// TIA Portal V15.1 export
// export: Created 2024-06-21T08:41:01.4306107Z, ExportSetting WithDefaults, DisplayName Totally Integrated Automation Portal, DisplayVersion V15.1 Update 5, DisplayName TIA Portal Openness, DisplayVersion V15.1 Update 5, DisplayName SINAMICS Startdrive Advanced, DisplayVersion V15.1, DisplayName G130, G150, S120, S150, SINAMICS MV, S210, DisplayVersion V15.1, DisplayName G110M, G120, G120C, G120D, G120P, DisplayVersion V15.1, DisplayName STEP 7 Professional, DisplayVersion V15.1 Update 5, DisplayName STEP 7 Safety, DisplayVersion V15.1, DisplayName WinCC Professional, DisplayVersion V15.1 Update 5, DisplayName SIMATIC Visualization Architect, DisplayVersion V15.1
FUNCTION_BLOCK "LModeSelector"   // FB1002, FBD
TITLE = LModeSelector
{ S7_Optimized_Access := 'FALSE' }
AUTHOR : VCC
FAMILY : Control
NAME : ModeSel
VERSION : 1.0
// ================================================================================
// This module handles that only one mode is selected in the modezon, it also 
// handle interlocking between the HMIs. Each modezone can have 5 HMI.
// ================================================================================
// stored: AutoNumber false, IsIECCheckEnabled false, SetENOAutomatically False, UDAEnableTagReadback false
   VAR_INPUT
      I_NumHMI { ExternalAccessible := 'False'; ExternalVisible := 'False'; ExternalWritable := 'False'} : Int;   // Number of HMI used in the modezon
      I_LockManualTime { ExternalAccessible := 'False'; ExternalVisible := 'False'; ExternalWritable := 'False'} : Int;   // The number of seconds that Lock Manual shall be active
      I_StartPB { ExternalAccessible := 'False'; ExternalVisible := 'False'; ExternalWritable := 'False'} : Bool;   // Summary of Start buttons
      I_AlarmResetPB { ExternalAccessible := 'False'; ExternalVisible := 'False'; ExternalWritable := 'False'} : Bool;   // Summary of Alarm reset buttons
      I_SafetyNotOk { ExternalAccessible := 'False'; ExternalVisible := 'False'; ExternalWritable := 'False'} : Bool;   // Safety is not ok
      I_FailSafeResetAck { ExternalAccessible := 'False'; ExternalVisible := 'False'; ExternalWritable := 'False'} : Bool;   // F_Ack_Op FB in safety program is requesting value 9 on FailSafeReset output
      I_FailSafeAckID { ExternalAccessible := 'False'; ExternalVisible := 'False'; ExternalWritable := 'False'} : Int;   // F_Ack ID
      I_AllHMIAutoSel { ExternalAccessible := 'False'; ExternalVisible := 'False'; ExternalWritable := 'False'} : Bool;   // All HMI to Auto Selected
      I_HMI1ForceMan { ExternalAccessible := 'False'; ExternalVisible := 'False'; ExternalWritable := 'False'} : Bool;   // Forced manual selected on HMI1
      I_HMI1SetPB { ExternalAccessible := 'False'; ExternalVisible := 'False'; ExternalWritable := 'False'} : Bool;   // Set PB activated on HMI1
      I_HMI1ResetPB { ExternalAccessible := 'False'; ExternalVisible := 'False'; ExternalWritable := 'False'} : Bool;   // Reset PB activated on HMI1
      I_HMI1StartPB { ExternalAccessible := 'False'; ExternalVisible := 'False'; ExternalWritable := 'False'} : Bool;   // Start PB activated on HMI1
      I_HMI1AlarmResetPB { ExternalAccessible := 'False'; ExternalVisible := 'False'; ExternalWritable := 'False'} : Bool;   // AlarmReset PB activated on HMI1
      I_HMI2ForceMan { ExternalAccessible := 'False'; ExternalVisible := 'False'; ExternalWritable := 'False'} : Bool;   // Forced manual selected on HMI2
      I_HMI2SetPB { ExternalAccessible := 'False'; ExternalVisible := 'False'; ExternalWritable := 'False'} : Bool;   // Set PB activated on HMI2
      I_HMI2ResetPB { ExternalAccessible := 'False'; ExternalVisible := 'False'; ExternalWritable := 'False'} : Bool;   // Reset PB activated on HMI2
      I_HMI2StartPB { ExternalAccessible := 'False'; ExternalVisible := 'False'; ExternalWritable := 'False'} : Bool;   // Start PB activated on HMI2
      I_HMI2AlarmResetPB { ExternalAccessible := 'False'; ExternalVisible := 'False'; ExternalWritable := 'False'} : Bool;   // AlarmReset PB activated on HMI2
      I_HMI3ForceMan { ExternalAccessible := 'False'; ExternalVisible := 'False'; ExternalWritable := 'False'} : Bool;   // Forced manual selected on HMI3
      I_HMI3SetPB { ExternalAccessible := 'False'; ExternalVisible := 'False'; ExternalWritable := 'False'} : Bool;   // Set PB activated on HMI3
      I_HMI3ResetPB { ExternalAccessible := 'False'; ExternalVisible := 'False'; ExternalWritable := 'False'} : Bool;   // Reset PB activated on HMI3
      I_HMI3StartPB { ExternalAccessible := 'False'; ExternalVisible := 'False'; ExternalWritable := 'False'} : Bool;   // Start PB activated on HMI
      I_HMI3AlarmResetPB { ExternalAccessible := 'False'; ExternalVisible := 'False'; ExternalWritable := 'False'} : Bool;   // AlarmReset PB activated on HMI3
      I_HMI4ForceMan { ExternalAccessible := 'False'; ExternalVisible := 'False'; ExternalWritable := 'False'} : Bool;   // Forced manual selected on HMI4
      I_HMI4SetPB { ExternalAccessible := 'False'; ExternalVisible := 'False'; ExternalWritable := 'False'} : Bool;   // Set PB activated on HMI4
      I_HMI4ResetPB { ExternalAccessible := 'False'; ExternalVisible := 'False'; ExternalWritable := 'False'} : Bool;   // Reset PB activated on HMI4
      I_HMI4StartPB { ExternalAccessible := 'False'; ExternalVisible := 'False'; ExternalWritable := 'False'} : Bool;   // Start PB activated on HMI4
      I_HMI4AlarmResetPB { ExternalAccessible := 'False'; ExternalVisible := 'False'; ExternalWritable := 'False'} : Bool;   // AlarmReset PB activated on HMI4
      I_HMI5ForceMan { ExternalAccessible := 'False'; ExternalVisible := 'False'; ExternalWritable := 'False'} : Bool;   // Forced manual selected on HMI5
      I_HMI5SetPB { ExternalAccessible := 'False'; ExternalVisible := 'False'; ExternalWritable := 'False'} : Bool;   // Set PB activated on HMI5
      I_HMI5ResetPB { ExternalAccessible := 'False'; ExternalVisible := 'False'; ExternalWritable := 'False'} : Bool;   // Reset PB activated on HMI5
      I_HMI5StartPB { ExternalAccessible := 'False'; ExternalVisible := 'False'; ExternalWritable := 'False'} : Bool;   // Start PB activated on HMI5
      I_HMI5AlarmResetPB { ExternalAccessible := 'False'; ExternalVisible := 'False'; ExternalWritable := 'False'} : Bool;   // AlarmReset PB activated on HMI5
   END_VAR
   VAR_OUTPUT
      O_AutoSel { ExternalAccessible := 'False'; ExternalVisible := 'False'; ExternalWritable := 'False'} : Bool;   // Auto selected
      O_AllAutoSel { ExternalAccessible := 'False'; ExternalVisible := 'False'; ExternalWritable := 'False'} : Bool;   // All objects in Auto selected
      O_StepSel { ExternalAccessible := 'False'; ExternalVisible := 'False'; ExternalWritable := 'False'} : Bool;   // Step selected
      O_HomeRunSel { ExternalAccessible := 'False'; ExternalVisible := 'False'; ExternalWritable := 'False'} : Bool;   // Homerun selected
      O_ManualSel { ExternalAccessible := 'False'; ExternalVisible := 'False'; ExternalWritable := 'False'} : Bool;   // Manual selected
      O_ForcedManActSel { ExternalAccessible := 'False'; ExternalVisible := 'False'; ExternalWritable := 'False'} : Bool;   // Forced manual selected
      O_PBSetSel { ExternalAccessible := 'False'; ExternalVisible := 'False'; ExternalWritable := 'False'} : Bool;   // Set selected
      O_PBResetSel { ExternalAccessible := 'False'; ExternalVisible := 'False'; ExternalWritable := 'False'} : Bool;   // Reset selected
      O_StartPBSel { ExternalAccessible := 'False'; ExternalVisible := 'False'; ExternalWritable := 'False'} : Bool;   // Start is activated
      O_AlarmResetPBSel { ExternalAccessible := 'False'; ExternalVisible := 'False'; ExternalWritable := 'False'} : Bool;   // Alarm reset is activated
      O_ResetTMSel { ExternalAccessible := 'False'; ExternalVisible := 'False'; ExternalWritable := 'False'} : Bool;   // Reset transport memory
      O_ResetSeqSel { ExternalAccessible := 'False'; ExternalVisible := 'False'; ExternalWritable := 'False'} : Bool;   // Reset squence
      O_CycleFinishedSel { ExternalAccessible := 'False'; ExternalVisible := 'False'; ExternalWritable := 'False'} : Bool;   // Cycle finished selected
      O_HomeRunRedoSel { ExternalAccessible := 'False'; ExternalVisible := 'False'; ExternalWritable := 'False'} : Bool;   // Redo after Homerun selected
      O_HomeRunWorkDoneSel { ExternalAccessible := 'False'; ExternalVisible := 'False'; ExternalWritable := 'False'} : Bool;   // WorkDone after Homerun selected
   END_VAR
   VAR_IN_OUT
      IO_FailsafeReset { ExternalAccessible := 'False'; ExternalVisible := 'False'; ExternalWritable := 'False'} : Int;   // Number to Failsafe to reset safety
   END_VAR
   VAR DB_SPECIFIC
      H_HMIHomeRunModeCmd : Word;   // Homerun Mode commands from HMI
      H_Anim : Word;   // Animation for HMI
      H_ActiveHMI : Int;   // Active HMI
      H_NameActiveHMI : String[25];   // Name of the Active HMI
      H_LockManTime : Int;   // Lock manual time
      H_HMI1ModeCmd : Word;   // Mode commands from HMI1
      H_HMI2ModeCmd : Word;   // Mode commands from HMI2
      H_HMI3ModeCmd : Word;   // Mode commands from HMI3
      H_HMI4ModeCmd : Word;   // Mode commands from HMI4
      H_HMI5ModeCmd : Word;   // Mode commands from HMI5. For operator panels, no S7_m_c
      HMI1AutoSel { ExternalAccessible := 'False'; ExternalVisible := 'False'; ExternalWritable := 'False'} : Bool;   // Auto selected on HMI1
      HMI1StepSel { ExternalAccessible := 'False'; ExternalVisible := 'False'; ExternalWritable := 'False'} : Bool;   // Step selected on HMI1
      HMI1HomeRunSel { ExternalAccessible := 'False'; ExternalVisible := 'False'; ExternalWritable := 'False'} : Bool;   // Homerun selected on HMI1
      HMI1ManualSel { ExternalAccessible := 'False'; ExternalVisible := 'False'; ExternalWritable := 'False'} : Bool;   // Manual selected on HMI1
      HMI1LockManual { ExternalAccessible := 'False'; ExternalVisible := 'False'; ExternalWritable := 'False'} : Bool;   // Lock manual for HMI1
      HMI1AllHMIAutoSel { ExternalAccessible := 'False'; ExternalVisible := 'False'; ExternalWritable := 'False'} : Bool;   // All HMI Auto selected on HMI1
      HMI1Start { ExternalAccessible := 'False'; ExternalVisible := 'False'; ExternalWritable := 'False'} : Bool;   // Start on HMI1
      HMI1AlarmReset { ExternalAccessible := 'False'; ExternalVisible := 'False'; ExternalWritable := 'False'} : Bool;   // AlarmReset on HMI1
      HMI1ResetTM { ExternalAccessible := 'False'; ExternalVisible := 'False'; ExternalWritable := 'False'} : Bool;   // Reset transport memory from HMI1
      HMI1ResetSeq { ExternalAccessible := 'False'; ExternalVisible := 'False'; ExternalWritable := 'False'} : Bool;   // Reset sequence from HMI1
      HMI1CycleFinished { ExternalAccessible := 'False'; ExternalVisible := 'False'; ExternalWritable := 'False'} : Bool;   // Cycle Finished from HMI1
      HMI1AlarmResetAck { ExternalAccessible := 'False'; ExternalVisible := 'False'; ExternalWritable := 'False'} : Bool;   // Alarm Reset acknowledge from HMI1
      HMI2AutoSel { ExternalAccessible := 'False'; ExternalVisible := 'False'; ExternalWritable := 'False'} : Bool;   // Auto selected on HMI2
      HMI2StepSel { ExternalAccessible := 'False'; ExternalVisible := 'False'; ExternalWritable := 'False'} : Bool;   // Step selected on HMI2
      HMI2HomeRunSel { ExternalAccessible := 'False'; ExternalVisible := 'False'; ExternalWritable := 'False'} : Bool;   // Homerun selected on HMI2
      HMI2ManualSel { ExternalAccessible := 'False'; ExternalVisible := 'False'; ExternalWritable := 'False'} : Bool;   // Manual selected on HMI2
      HMI2LockManual { ExternalAccessible := 'False'; ExternalVisible := 'False'; ExternalWritable := 'False'} : Bool;   // Lock manual for HMI2
      HMI2AllHMIAutoSel { ExternalAccessible := 'False'; ExternalVisible := 'False'; ExternalWritable := 'False'} : Bool;   // All HMI Auto selected on HMI2
      HMI2Start { ExternalAccessible := 'False'; ExternalVisible := 'False'; ExternalWritable := 'False'} : Bool;   // Start on HMI2
      HMI2AlarmReset { ExternalAccessible := 'False'; ExternalVisible := 'False'; ExternalWritable := 'False'} : Bool;   // AlarmReset on HMI2
      HMI2ResetTM { ExternalAccessible := 'False'; ExternalVisible := 'False'; ExternalWritable := 'False'} : Bool;   // Reset transport memory from HMI2
      HMI2ResetSeq { ExternalAccessible := 'False'; ExternalVisible := 'False'; ExternalWritable := 'False'} : Bool;   // Reset sequence from HMI2
      HMI2CycleFinished { ExternalAccessible := 'False'; ExternalVisible := 'False'; ExternalWritable := 'False'} : Bool;   // Cycle Finished from HMI2
      HMI2AlarmResetAck { ExternalAccessible := 'False'; ExternalVisible := 'False'; ExternalWritable := 'False'} : Bool;   // Alarm Reset acknowledge from HMI2
      HMI3AutoSel { ExternalAccessible := 'False'; ExternalVisible := 'False'; ExternalWritable := 'False'} : Bool;   // Auto selected on HMI3
      HMI3StepSel { ExternalAccessible := 'False'; ExternalVisible := 'False'; ExternalWritable := 'False'} : Bool;   // Step selected on HMI3
      HMI3HomeRunSel { ExternalAccessible := 'False'; ExternalVisible := 'False'; ExternalWritable := 'False'} : Bool;   // Homerun selected on HMI3
      HMI3ManualSel { ExternalAccessible := 'False'; ExternalVisible := 'False'; ExternalWritable := 'False'} : Bool;   // Manual selected on HMI3
      HMI3LockManual { ExternalAccessible := 'False'; ExternalVisible := 'False'; ExternalWritable := 'False'} : Bool;   // Lock manual for HMI3
      HMI3AllHMIAutoSel { ExternalAccessible := 'False'; ExternalVisible := 'False'; ExternalWritable := 'False'} : Bool;   // All HMI Auto selected on HMI3
      HMI3Start { ExternalAccessible := 'False'; ExternalVisible := 'False'; ExternalWritable := 'False'} : Bool;   // Start on HMI3
      HMI3AlarmReset { ExternalAccessible := 'False'; ExternalVisible := 'False'; ExternalWritable := 'False'} : Bool;   // AlarmReset on HMI3
      HMI3ResetTM { ExternalAccessible := 'False'; ExternalVisible := 'False'; ExternalWritable := 'False'} : Bool;   // Reset transport memory from HMI3
      HMI3ResetSeq { ExternalAccessible := 'False'; ExternalVisible := 'False'; ExternalWritable := 'False'} : Bool;   // Reset sequence from HMI3
      HMI3CycleFinished { ExternalAccessible := 'False'; ExternalVisible := 'False'; ExternalWritable := 'False'} : Bool;   // Cycle Finished from HMI3
      HMI3AlarmResetAck { ExternalAccessible := 'False'; ExternalVisible := 'False'; ExternalWritable := 'False'} : Bool;   // Alarm Reset acknowledge from 3
      HMI4AutoSel { ExternalAccessible := 'False'; ExternalVisible := 'False'; ExternalWritable := 'False'} : Bool;   // Auto selected on HMI4
      HMI4StepSel { ExternalAccessible := 'False'; ExternalVisible := 'False'; ExternalWritable := 'False'} : Bool;   // Step selected on HMI4
      HMI4HomeRunSel { ExternalAccessible := 'False'; ExternalVisible := 'False'; ExternalWritable := 'False'} : Bool;   // Homerun selected on HMI4
      HMI4ManualSel { ExternalAccessible := 'False'; ExternalVisible := 'False'; ExternalWritable := 'False'} : Bool;   // Manual selected on HMI4
      HMI4LockManual { ExternalAccessible := 'False'; ExternalVisible := 'False'; ExternalWritable := 'False'} : Bool;   // Lock manual for HMI4
      HMI4AllHMIAutoSel { ExternalAccessible := 'False'; ExternalVisible := 'False'; ExternalWritable := 'False'} : Bool;   // All HMI Auto selected on HMI4
      HMI4Start { ExternalAccessible := 'False'; ExternalVisible := 'False'; ExternalWritable := 'False'} : Bool;   // Start on HMI4
      HMI4AlarmReset { ExternalAccessible := 'False'; ExternalVisible := 'False'; ExternalWritable := 'False'} : Bool;   // AlarmReset on HMI4
      HMI4ResetTM { ExternalAccessible := 'False'; ExternalVisible := 'False'; ExternalWritable := 'False'} : Bool;   // Reset transport memory from HMI4
      HMI4ResetSeq { ExternalAccessible := 'False'; ExternalVisible := 'False'; ExternalWritable := 'False'} : Bool;   // Reset sequence from HMI4
      HMI4CycleFinished { ExternalAccessible := 'False'; ExternalVisible := 'False'; ExternalWritable := 'False'} : Bool;   // Cycle Finished from HMI4
      HMI4AlarmResetAck { ExternalAccessible := 'False'; ExternalVisible := 'False'; ExternalWritable := 'False'} : Bool;   // Alarm Reset acknowledge from HMI4
      HMI5AutoSel { ExternalAccessible := 'False'; ExternalVisible := 'False'; ExternalWritable := 'False'} : Bool;   // Auto selected on HMI5
      HMI5StepSel { ExternalAccessible := 'False'; ExternalVisible := 'False'; ExternalWritable := 'False'} : Bool;   // Step selected on HMI5
      HMI5HomeRunSel { ExternalAccessible := 'False'; ExternalVisible := 'False'; ExternalWritable := 'False'} : Bool;   // Homerun selected on HMI5
      HMI5ManualSel { ExternalAccessible := 'False'; ExternalVisible := 'False'; ExternalWritable := 'False'} : Bool;   // Manual selected on HMI5
      HMI5LockManual { ExternalAccessible := 'False'; ExternalVisible := 'False'; ExternalWritable := 'False'} : Bool;   // Lock manual for HMI5
      HMI5AllHMIAutoSel { ExternalAccessible := 'False'; ExternalVisible := 'False'; ExternalWritable := 'False'} : Bool;   // All HMI Auto selected on HMI5
      HMI5Start { ExternalAccessible := 'False'; ExternalVisible := 'False'; ExternalWritable := 'False'} : Bool;   // Start on HMI5
      HMI5AlarmReset { ExternalAccessible := 'False'; ExternalVisible := 'False'; ExternalWritable := 'False'} : Bool;   // AlarmReset on HMI5
      HMI5ResetTM { ExternalAccessible := 'False'; ExternalVisible := 'False'; ExternalWritable := 'False'} : Bool;   // Reset transport memory from HMI5
      HMI5ResetSeq { ExternalAccessible := 'False'; ExternalVisible := 'False'; ExternalWritable := 'False'} : Bool;   // Reset sequence from HMI5
      HMI5CycleFinished { ExternalAccessible := 'False'; ExternalVisible := 'False'; ExternalWritable := 'False'} : Bool;   // Cycle Finished from HMI5
      HMI5AlarmResetAck { ExternalAccessible := 'False'; ExternalVisible := 'False'; ExternalWritable := 'False'} : Bool;   // Alarm Reset acknowledge from HMI5
      HMIHomeRunRedo { ExternalAccessible := 'False'; ExternalVisible := 'False'; ExternalWritable := 'False'} : Bool;   // Redo after homerun from HMI
      HMIHomeRunWorkDone { ExternalAccessible := 'False'; ExternalVisible := 'False'; ExternalWritable := 'False'} : Bool;   // WorkDone after homerun from HMI
      LockManualTimeout { ExternalAccessible := 'False'; ExternalVisible := 'False'; ExternalWritable := 'False'} : Bool;   // Lock manual button timeout
      AllHmiAutoSel { ExternalAccessible := 'False'; ExternalVisible := 'False'; ExternalWritable := 'False'} : Bool;   // All Hmi Auto selected
      AlarmResetPBSel { ExternalAccessible := 'False'; ExternalVisible := 'False'; ExternalWritable := 'False'} : Bool;   // Alarm reset is activated
      AlarmResetPBSelReset { ExternalAccessible := 'False'; ExternalVisible := 'False'; ExternalWritable := 'False'} : Bool;   // Reset AlarmResetPBSel after predefined time
      AlarmResetPBSelResetPE { ExternalAccessible := 'False'; ExternalVisible := 'False'; ExternalWritable := 'False'} : Bool;   // Positive edge of AlarmResetPbSelReset
      FailSafeReset6Pulse { ExternalAccessible := 'False'; ExternalVisible := 'False'; ExternalWritable := 'False'} : Bool;   // Pulse to set value 6 on FailSafeReset Output
      FailSafeReset9Pulse { ExternalAccessible := 'False'; ExternalVisible := 'False'; ExternalWritable := 'False'} : Bool;   // Pulse to set value 9 on FailSafeReset Output
      ResetAlarmAckMemPulse { ExternalAccessible := 'False'; ExternalVisible := 'False'; ExternalWritable := 'False'} : Bool;   // Pulse to reset AlarmResetAckMem on negative edge of I_FailSafeResetAck
      AlarmResetAckMem { ExternalAccessible := 'False'; ExternalVisible := 'False'; ExternalWritable := 'False'} : Bool;   // memory : Pushbutton AlarmResetAck has been pushed on HMI
      StartPBSel { ExternalAccessible := 'False'; ExternalVisible := 'False'; ExternalWritable := 'False'} : Bool;   // Summary of the Start push buttons
      AutoSel { ExternalAccessible := 'False'; ExternalVisible := 'False'; ExternalWritable := 'False'} : Bool;   // Auto selected
      HMIStartPE { ExternalAccessible := 'False'; ExternalVisible := 'False'; ExternalWritable := 'False'} : Bool;   // Positive edge on start button from HMI
      HMIResetTMPE { ExternalAccessible := 'False'; ExternalVisible := 'False'; ExternalWritable := 'False'} : Bool;   // Positive edge on ResetTM button from HMI
      HMIResetSeqPE { ExternalAccessible := 'False'; ExternalVisible := 'False'; ExternalWritable := 'False'} : Bool;   // Positive edge on ResetSeq button from HMI
      HMIAlarmResetAckPE { ExternalAccessible := 'False'; ExternalVisible := 'False'; ExternalWritable := 'False'} : Bool;   // Positive edge on AlarmResetAck button from HMI
      HMILockManualPE { ExternalAccessible := 'False'; ExternalVisible := 'False'; ExternalWritable := 'False'} : Bool;   // Positive edge on LockManual button from HMI
      PBSetSel { ExternalAccessible := 'False'; ExternalVisible := 'False'; ExternalWritable := 'False'} : Bool;   // Set selected
      PBResetSel { ExternalAccessible := 'False'; ExternalVisible := 'False'; ExternalWritable := 'False'} : Bool;   // Reset selected
      CheckHMIActive { ExternalAccessible := 'False'; ExternalVisible := 'False'; ExternalWritable := 'False'} : Bool;   // Check Active HMI
      FailsafeReset { ExternalAccessible := 'False'; ExternalVisible := 'False'; ExternalWritable := 'False'} : Int;   // Number to Failsafe to reset safety
      ActiveHMI { ExternalAccessible := 'False'; ExternalVisible := 'False'; ExternalWritable := 'False'} : Int;   // Help memory for Active HMI
      LockManualSec { ExternalAccessible := 'False'; ExternalVisible := 'False'; ExternalWritable := 'False'} : DInt;   // Lock manual on for xxx milliesec
      LockManualMillieSec { ExternalAccessible := 'False'; ExternalVisible := 'False'; ExternalWritable := 'False'} : DInt;   // Converted value
      TimerLockManValue { ExternalAccessible := 'False'; ExternalVisible := 'False'; ExternalWritable := 'False'} : DInt;   // Timer value
   END_VAR
   VAR
      TimerLockMan { ExternalAccessible := 'False'; ExternalVisible := 'False'; ExternalWritable := 'False'; S7_SetPoint := 'True'} : "LTimer";   // Timer on Lock manual
      TimerAlarmResetPB { ExternalAccessible := 'False'; ExternalVisible := 'False'; ExternalWritable := 'False'; S7_SetPoint := 'True'} : "LTimer";   // Timer on alarm reset
   END_VAR
   VAR DB_SPECIFIC
      CheckActiveHMI { ExternalAccessible := 'False'; ExternalVisible := 'False'; ExternalWritable := 'False'; S7_SetPoint := 'True'} : TP_TIME;   // Timer
      CheckActiveHMI_1 { ExternalAccessible := 'False'; ExternalVisible := 'False'; ExternalWritable := 'False'; S7_SetPoint := 'True'} : TP_TIME;   // Timer
      CheckActiveHMI_2 { ExternalAccessible := 'False'; ExternalVisible := 'False'; ExternalWritable := 'False'; S7_SetPoint := 'True'} : TON_TIME;   // Timer
      CheckActiveHMI_3 { ExternalAccessible := 'False'; ExternalVisible := 'False'; ExternalWritable := 'False'; S7_SetPoint := 'True'} : TON_TIME;   // Timer
   END_VAR
   VAR_TEMP
      PHMI1AutoSel : Bool;   // Pulse Auto selected HMI1
      PHMI2AutoSel : Bool;   // Pulse Auto selected HMI2
      PHMI3AutoSel : Bool;   // Pulse Auto selected HMI3
      PHMI4AutoSel : Bool;   // Pulse Auto selected HMI4
      PHMI5AutoSel : Bool;   // Pulse Auto selected HMI5
      LockManualTime : Int;   // Lock manual time
      LockManualTimeInt : Int;   // Lock manual time
      LockManualTimeDInt : DInt;   // Lock manual time
   END_VAR
   VAR_TEMP   // added for the SCL form of the ladder/FBD networks
      _w1 : Bool;
      _w2 : Bool;
      _w3 : Bool;
      _w4 : Bool;
      _w5 : Bool;
   END_VAR
BEGIN

REGION Network 1: **** 1 - Inputs **** Extract the modeselection from HMI 1
   // Extract the modeselection from HMI 1
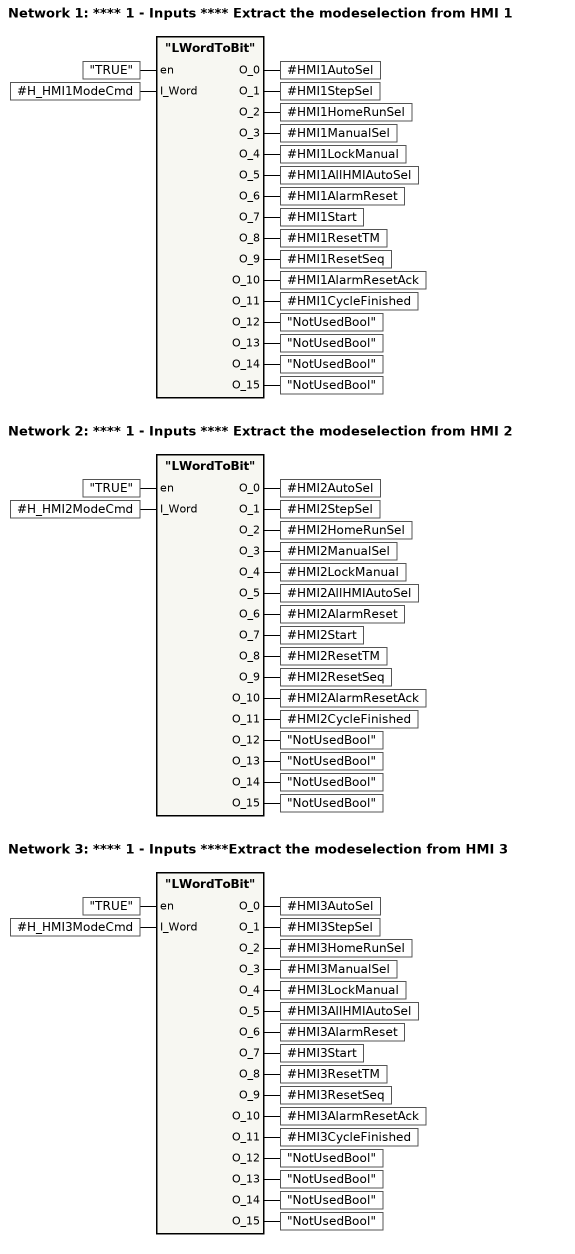
   IF "TRUE" THEN
       "LWordToBit"(I_Word := #H_HMI1ModeCmd,
                    O_0 => #HMI1AutoSel,
                    O_1 => #HMI1StepSel,
                    O_2 => #HMI1HomeRunSel,
                    O_3 => #HMI1ManualSel,
                    O_4 => #HMI1LockManual,
                    O_5 => #HMI1AllHMIAutoSel,
                    O_6 => #HMI1AlarmReset,
                    O_7 => #HMI1Start,
                    O_8 => #HMI1ResetTM,
                    O_9 => #HMI1ResetSeq,
                    O_10 => #HMI1AlarmResetAck,
                    O_11 => #HMI1CycleFinished,
                    O_12 => "NotUsedBool",
                    O_13 => "NotUsedBool",
                    O_14 => "NotUsedBool",
                    O_15 => "NotUsedBool");
   END_IF;
END_REGION

REGION Network 2: **** 1 - Inputs **** Extract the modeselection from HMI 2
   // Extract the modeselection from HMI 2
   IF "TRUE" THEN
       "LWordToBit"(I_Word := #H_HMI2ModeCmd,
                    O_0 => #HMI2AutoSel,
                    O_1 => #HMI2StepSel,
                    O_2 => #HMI2HomeRunSel,
                    O_3 => #HMI2ManualSel,
                    O_4 => #HMI2LockManual,
                    O_5 => #HMI2AllHMIAutoSel,
                    O_6 => #HMI2AlarmReset,
                    O_7 => #HMI2Start,
                    O_8 => #HMI2ResetTM,
                    O_9 => #HMI2ResetSeq,
                    O_10 => #HMI2AlarmResetAck,
                    O_11 => #HMI2CycleFinished,
                    O_12 => "NotUsedBool",
                    O_13 => "NotUsedBool",
                    O_14 => "NotUsedBool",
                    O_15 => "NotUsedBool");
   END_IF;
END_REGION

REGION Network 3: **** 1 - Inputs ****Extract the modeselection from HMI 3
   // Extract the modeselection from HMI 3
   IF "TRUE" THEN
       "LWordToBit"(I_Word := #H_HMI3ModeCmd,
                    O_0 => #HMI3AutoSel,
                    O_1 => #HMI3StepSel,
                    O_2 => #HMI3HomeRunSel,
                    O_3 => #HMI3ManualSel,
                    O_4 => #HMI3LockManual,
                    O_5 => #HMI3AllHMIAutoSel,
                    O_6 => #HMI3AlarmReset,
                    O_7 => #HMI3Start,
                    O_8 => #HMI3ResetTM,
                    O_9 => #HMI3ResetSeq,
                    O_10 => #HMI3AlarmResetAck,
                    O_11 => #HMI3CycleFinished,
                    O_12 => "NotUsedBool",
                    O_13 => "NotUsedBool",
                    O_14 => "NotUsedBool",
                    O_15 => "NotUsedBool");
   END_IF;
END_REGION

REGION Network 4: **** 1 - Inputs **** Extract the modeselection from HMI 4
   // Extract the modeselection from HMI 4
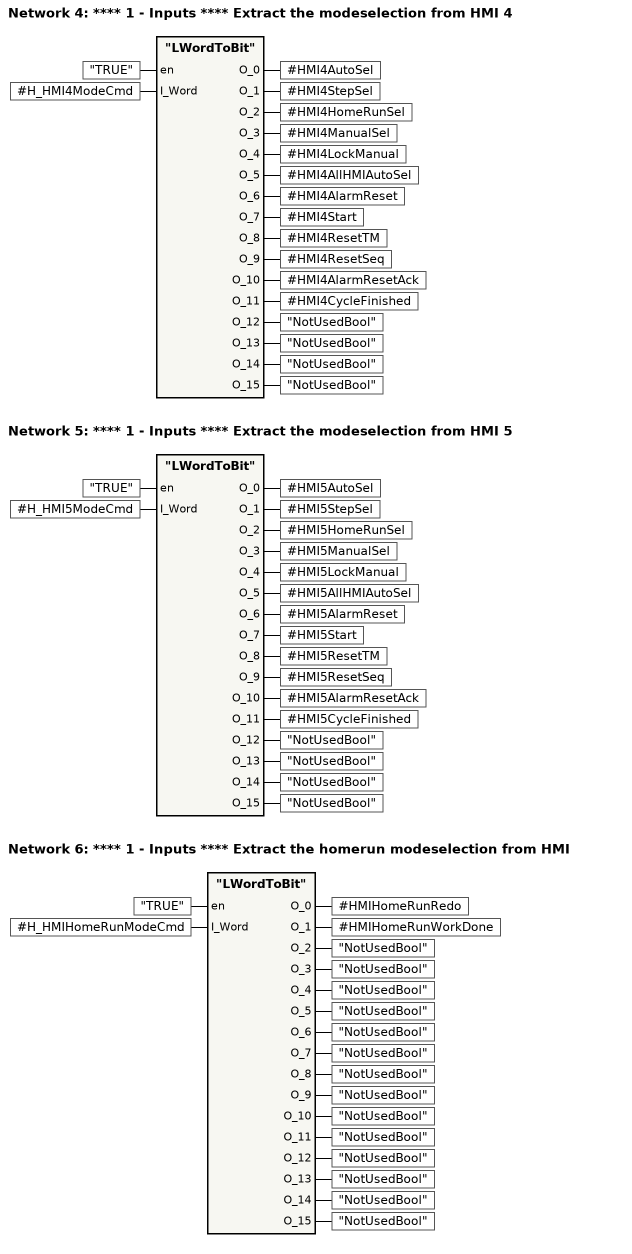
   IF "TRUE" THEN
       "LWordToBit"(I_Word := #H_HMI4ModeCmd,
                    O_0 => #HMI4AutoSel,
                    O_1 => #HMI4StepSel,
                    O_2 => #HMI4HomeRunSel,
                    O_3 => #HMI4ManualSel,
                    O_4 => #HMI4LockManual,
                    O_5 => #HMI4AllHMIAutoSel,
                    O_6 => #HMI4AlarmReset,
                    O_7 => #HMI4Start,
                    O_8 => #HMI4ResetTM,
                    O_9 => #HMI4ResetSeq,
                    O_10 => #HMI4AlarmResetAck,
                    O_11 => #HMI4CycleFinished,
                    O_12 => "NotUsedBool",
                    O_13 => "NotUsedBool",
                    O_14 => "NotUsedBool",
                    O_15 => "NotUsedBool");
   END_IF;
END_REGION

REGION Network 5: **** 1 - Inputs **** Extract the modeselection from HMI 5
   // Extract the modeselection from HMI 5
   IF "TRUE" THEN
       "LWordToBit"(I_Word := #H_HMI5ModeCmd,
                    O_0 => #HMI5AutoSel,
                    O_1 => #HMI5StepSel,
                    O_2 => #HMI5HomeRunSel,
                    O_3 => #HMI5ManualSel,
                    O_4 => #HMI5LockManual,
                    O_5 => #HMI5AllHMIAutoSel,
                    O_6 => #HMI5AlarmReset,
                    O_7 => #HMI5Start,
                    O_8 => #HMI5ResetTM,
                    O_9 => #HMI5ResetSeq,
                    O_10 => #HMI5AlarmResetAck,
                    O_11 => #HMI5CycleFinished,
                    O_12 => "NotUsedBool",
                    O_13 => "NotUsedBool",
                    O_14 => "NotUsedBool",
                    O_15 => "NotUsedBool");
   END_IF;
END_REGION

REGION Network 6: **** 1 - Inputs **** Extract the homerun modeselection from HMI
   // Extract the homerun modeselection from HMI
   IF "TRUE" THEN
       "LWordToBit"(I_Word := #H_HMIHomeRunModeCmd,
                    O_0 => #HMIHomeRunRedo,
                    O_1 => #HMIHomeRunWorkDone,
                    O_2 => "NotUsedBool",
                    O_3 => "NotUsedBool",
                    O_4 => "NotUsedBool",
                    O_5 => "NotUsedBool",
                    O_6 => "NotUsedBool",
                    O_7 => "NotUsedBool",
                    O_8 => "NotUsedBool",
                    O_9 => "NotUsedBool",
                    O_10 => "NotUsedBool",
                    O_11 => "NotUsedBool",
                    O_12 => "NotUsedBool",
                    O_13 => "NotUsedBool",
                    O_14 => "NotUsedBool",
                    O_15 => "NotUsedBool");
   END_IF;
END_REGION

REGION Network 7: **** 1 - Inputs **** All HMI Auto selected
   // All HMI Auto selected
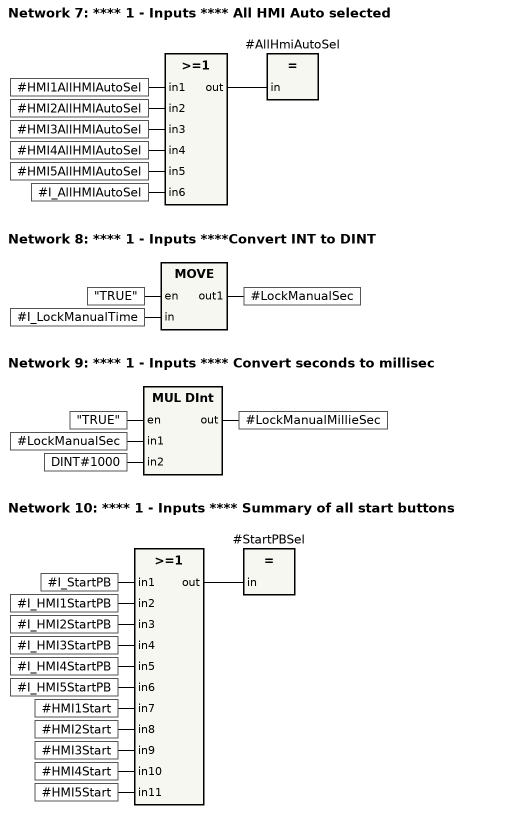
   #AllHmiAutoSel := #HMI1AllHMIAutoSel OR #HMI2AllHMIAutoSel OR #HMI3AllHMIAutoSel OR #HMI4AllHMIAutoSel OR #HMI5AllHMIAutoSel OR #I_AllHMIAutoSel;
END_REGION

REGION Network 8: **** 1 - Inputs ****Convert INT to DINT
   // Convert INT to DINT
   IF "TRUE" THEN #LockManualSec := #I_LockManualTime; END_IF;
END_REGION

REGION Network 9: **** 1 - Inputs **** Convert seconds to millisec
   // Convert seconds to millisec
   IF "TRUE" THEN #LockManualMillieSec := #LockManualSec * DINT#1000; END_IF;
END_REGION

REGION Network 10: **** 1 - Inputs **** Summary of all start buttons
   // Summary of all start buttons
   #StartPBSel := #I_StartPB OR #I_HMI1StartPB OR #I_HMI2StartPB OR #I_HMI3StartPB OR #I_HMI4StartPB OR #I_HMI5StartPB OR #HMI1Start OR #HMI2Start OR #HMI3Start OR #HMI4Start OR #HMI5Start;
END_REGION

REGION Network 11: **** 1 - Inputs **** Reset Start button from HMI
   // Reset Start button from HMI
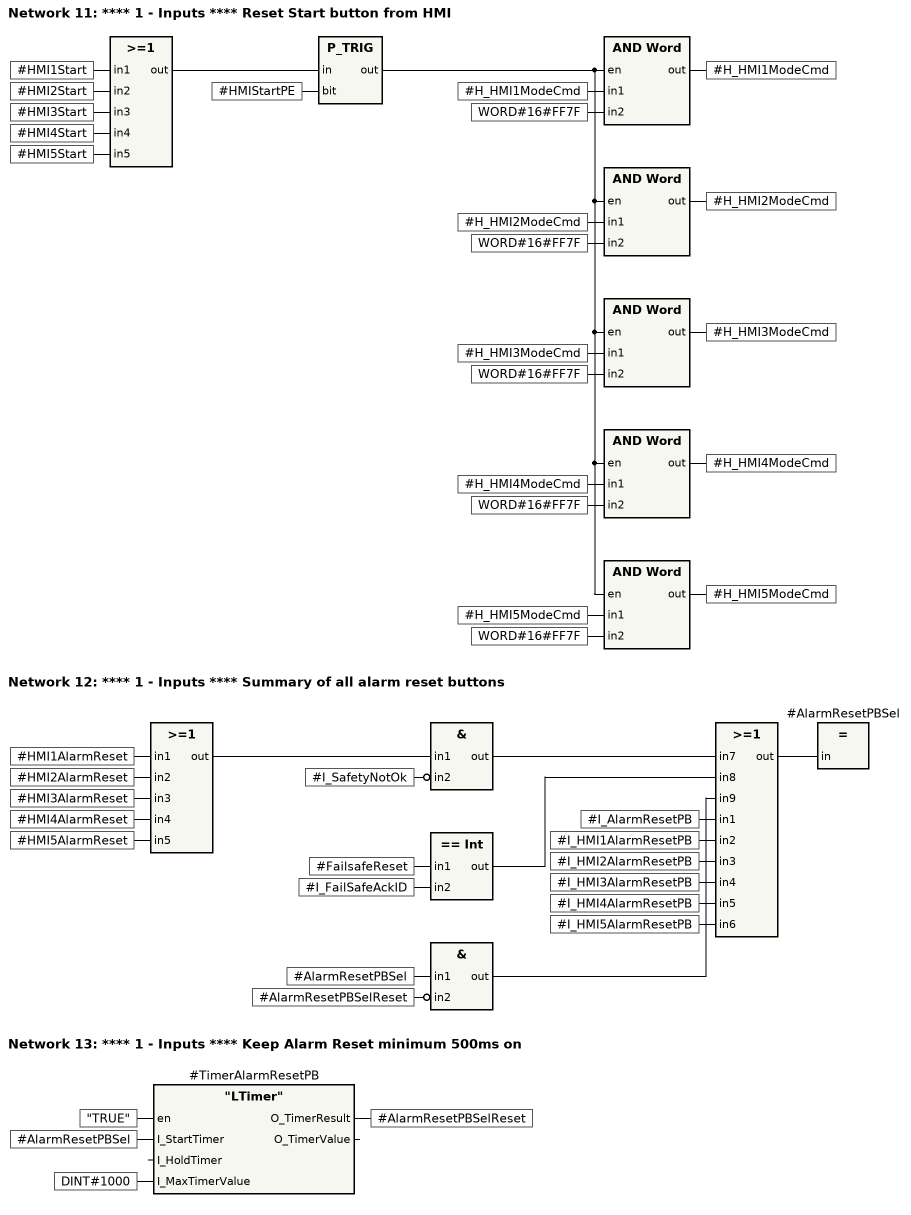
   #_w1 := #HMI1Start OR #HMI2Start OR #HMI3Start OR #HMI4Start OR #HMI5Start;
   #_w2 := #_w1 AND NOT #HMIStartPE;   // rising edge
   #HMIStartPE := #_w1;
   IF #_w2 THEN
       #H_HMI1ModeCmd := #H_HMI1ModeCmd AND WORD#16#FF7F;
       #H_HMI2ModeCmd := #H_HMI2ModeCmd AND WORD#16#FF7F;
       #H_HMI3ModeCmd := #H_HMI3ModeCmd AND WORD#16#FF7F;
       #H_HMI4ModeCmd := #H_HMI4ModeCmd AND WORD#16#FF7F;
       #H_HMI5ModeCmd := #H_HMI5ModeCmd AND WORD#16#FF7F;
   END_IF;
END_REGION

REGION Network 12: **** 1 - Inputs **** Summary of all alarm reset buttons
   // Summary of all alarm reset buttons
   #AlarmResetPBSel := ((#HMI1AlarmReset OR #HMI2AlarmReset OR #HMI3AlarmReset OR #HMI4AlarmReset OR #HMI5AlarmReset) AND NOT #I_SafetyNotOk) OR (#FailsafeReset = #I_FailSafeAckID) OR (#AlarmResetPBSel AND NOT #AlarmResetPBSelReset) OR #I_AlarmResetPB OR #I_HMI1AlarmResetPB OR #I_HMI2AlarmResetPB OR #I_HMI3AlarmResetPB OR #I_HMI4AlarmResetPB OR #I_HMI5AlarmResetPB;
END_REGION

REGION Network 13: **** 1 - Inputs **** Keep Alarm Reset minimum 500ms on
   // Keep Alarm Reset minimum 500ms on
   IF "TRUE" THEN
       #TimerAlarmResetPB(I_StartTimer := #AlarmResetPBSel,   // "LTimer"
                          I_MaxTimerValue := DINT#1000,
                          O_TimerResult => #AlarmResetPBSelReset);
   END_IF;
END_REGION

REGION Network 14: **** 1 - Inputs **** Reset AlarmResetPb from HMI
   // Reset AlarmResetPb from HMI
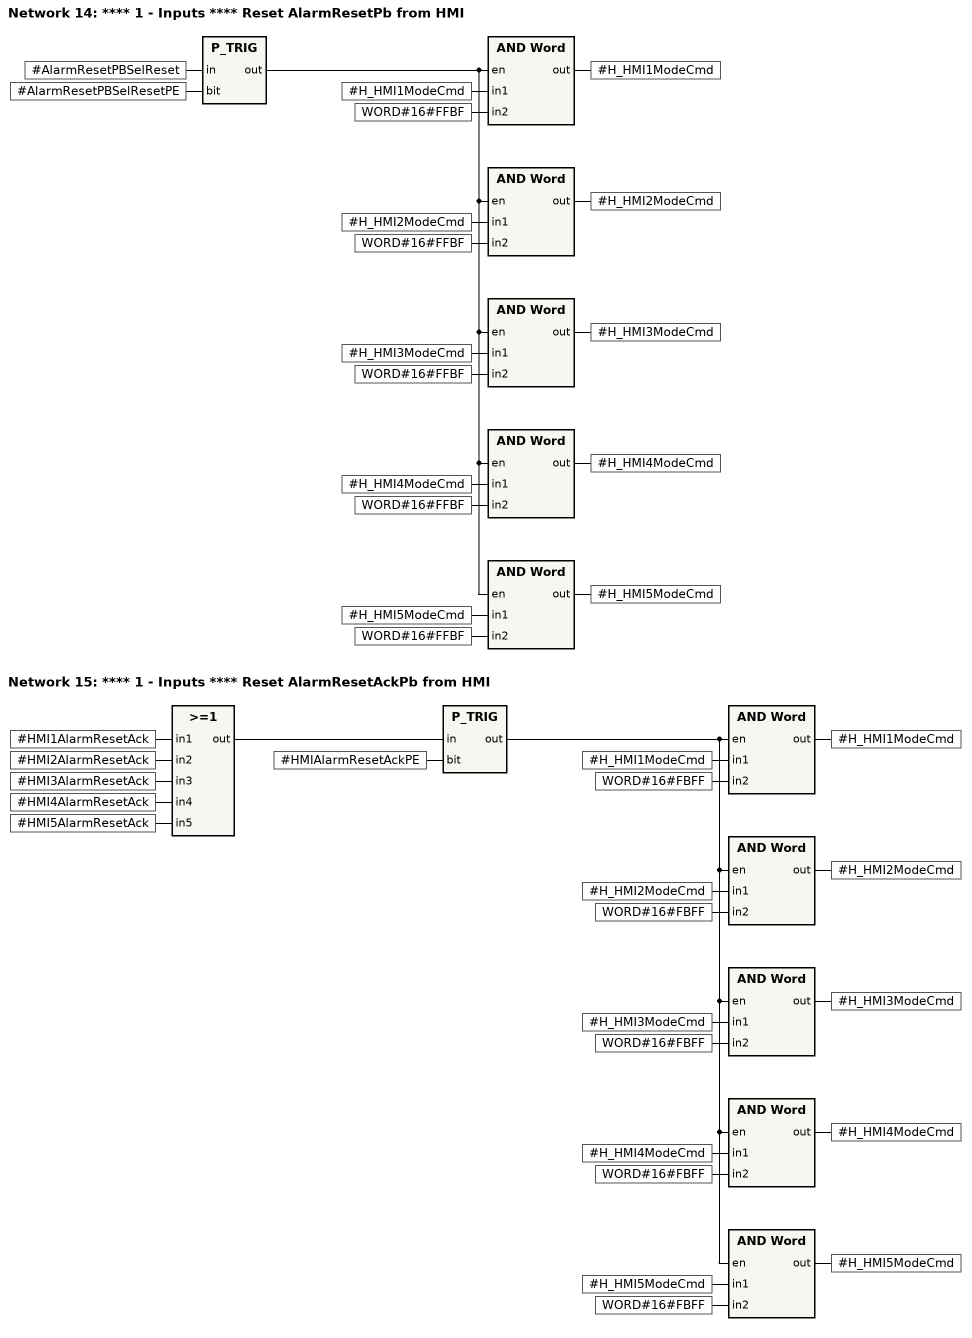
   #_w1 := #AlarmResetPBSelReset AND NOT #AlarmResetPBSelResetPE;   // rising edge
   #AlarmResetPBSelResetPE := #AlarmResetPBSelReset;
   IF #_w1 THEN
       #H_HMI1ModeCmd := #H_HMI1ModeCmd AND WORD#16#FFBF;
       #H_HMI2ModeCmd := #H_HMI2ModeCmd AND WORD#16#FFBF;
       #H_HMI3ModeCmd := #H_HMI3ModeCmd AND WORD#16#FFBF;
       #H_HMI4ModeCmd := #H_HMI4ModeCmd AND WORD#16#FFBF;
       #H_HMI5ModeCmd := #H_HMI5ModeCmd AND WORD#16#FFBF;
   END_IF;
END_REGION

REGION Network 15: **** 1 - Inputs **** Reset AlarmResetAckPb from HMI
   // Reset AlarmResetAckPb from HMI
   #_w1 := #HMI1AlarmResetAck OR #HMI2AlarmResetAck OR #HMI3AlarmResetAck OR #HMI4AlarmResetAck OR #HMI5AlarmResetAck;
   #_w2 := #_w1 AND NOT #HMIAlarmResetAckPE;   // rising edge
   #HMIAlarmResetAckPE := #_w1;
   IF #_w2 THEN
       #H_HMI1ModeCmd := #H_HMI1ModeCmd AND WORD#16#FBFF;
       #H_HMI2ModeCmd := #H_HMI2ModeCmd AND WORD#16#FBFF;
       #H_HMI3ModeCmd := #H_HMI3ModeCmd AND WORD#16#FBFF;
       #H_HMI4ModeCmd := #H_HMI4ModeCmd AND WORD#16#FBFF;
       #H_HMI5ModeCmd := #H_HMI5ModeCmd AND WORD#16#FBFF;
   END_IF;
END_REGION

REGION Network 16: **** 1 - Inputs **** Reset ResetTM button from HMI
   // Reset ResetTM button from HMI
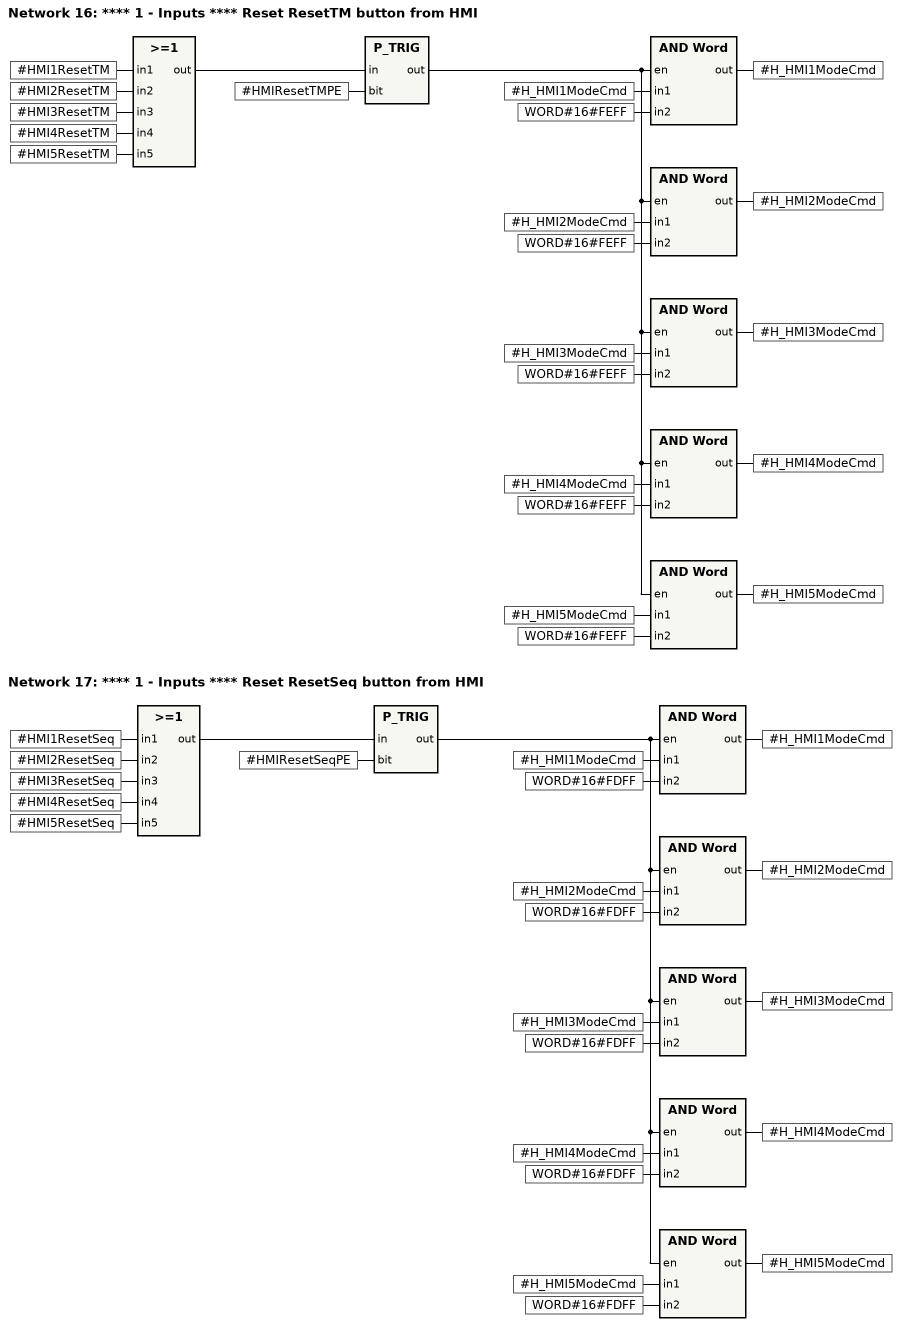
   #_w1 := #HMI1ResetTM OR #HMI2ResetTM OR #HMI3ResetTM OR #HMI4ResetTM OR #HMI5ResetTM;
   #_w2 := #_w1 AND NOT #HMIResetTMPE;   // rising edge
   #HMIResetTMPE := #_w1;
   IF #_w2 THEN
       #H_HMI1ModeCmd := #H_HMI1ModeCmd AND WORD#16#FEFF;
       #H_HMI2ModeCmd := #H_HMI2ModeCmd AND WORD#16#FEFF;
       #H_HMI3ModeCmd := #H_HMI3ModeCmd AND WORD#16#FEFF;
       #H_HMI4ModeCmd := #H_HMI4ModeCmd AND WORD#16#FEFF;
       #H_HMI5ModeCmd := #H_HMI5ModeCmd AND WORD#16#FEFF;
   END_IF;
END_REGION

REGION Network 17: **** 1 - Inputs **** Reset ResetSeq button from HMI
   // Reset ResetSeq button from HMI
   #_w1 := #HMI1ResetSeq OR #HMI2ResetSeq OR #HMI3ResetSeq OR #HMI4ResetSeq OR #HMI5ResetSeq;
   #_w2 := #_w1 AND NOT #HMIResetSeqPE;   // rising edge
   #HMIResetSeqPE := #_w1;
   IF #_w2 THEN
       #H_HMI1ModeCmd := #H_HMI1ModeCmd AND WORD#16#FDFF;
       #H_HMI2ModeCmd := #H_HMI2ModeCmd AND WORD#16#FDFF;
       #H_HMI3ModeCmd := #H_HMI3ModeCmd AND WORD#16#FDFF;
       #H_HMI4ModeCmd := #H_HMI4ModeCmd AND WORD#16#FDFF;
       #H_HMI5ModeCmd := #H_HMI5ModeCmd AND WORD#16#FDFF;
   END_IF;
END_REGION

REGION Network 18: **** 1 - Inputs **** Reset LockManual button from HMI
   // Reset LockManual button from HMI
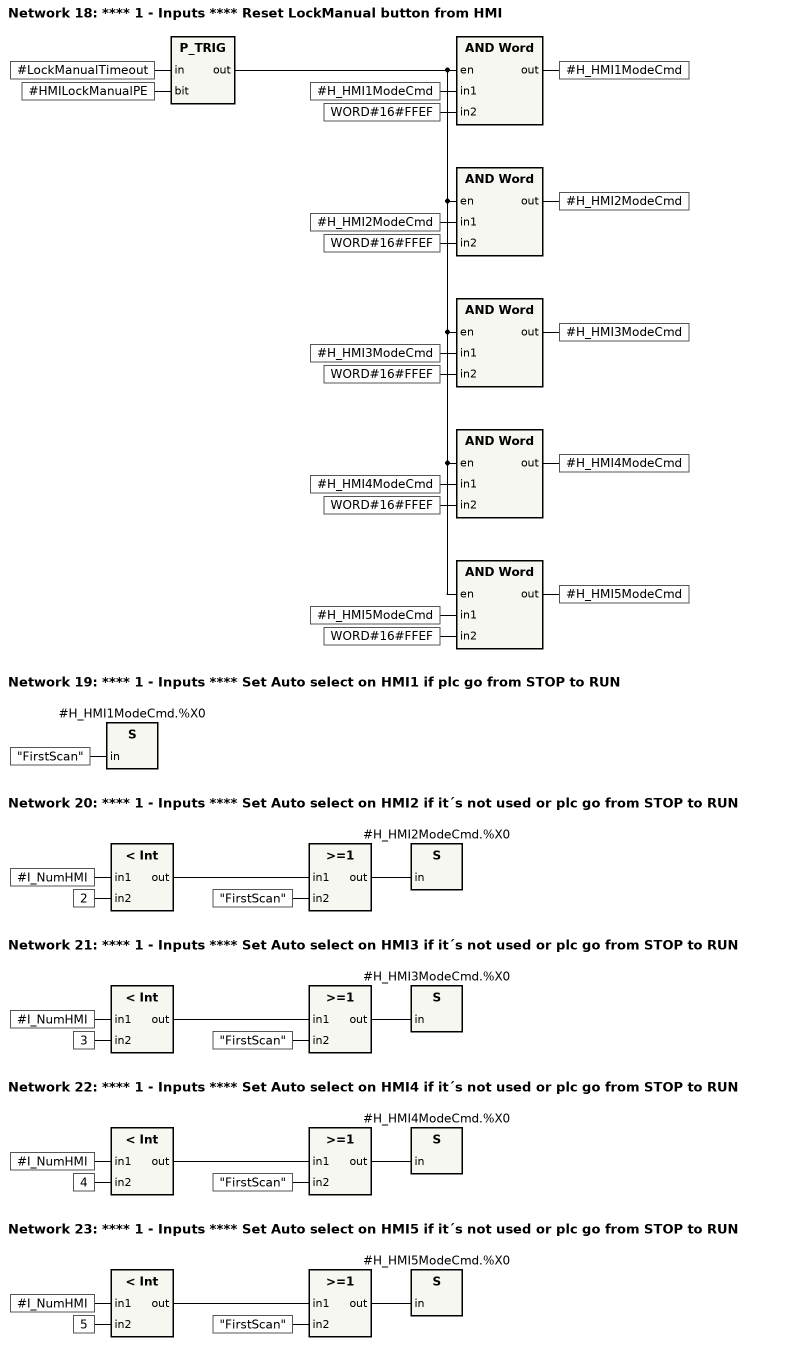
   #_w1 := #LockManualTimeout AND NOT #HMILockManualPE;   // rising edge
   #HMILockManualPE := #LockManualTimeout;
   IF #_w1 THEN
       #H_HMI1ModeCmd := #H_HMI1ModeCmd AND WORD#16#FFEF;
       #H_HMI2ModeCmd := #H_HMI2ModeCmd AND WORD#16#FFEF;
       #H_HMI3ModeCmd := #H_HMI3ModeCmd AND WORD#16#FFEF;
       #H_HMI4ModeCmd := #H_HMI4ModeCmd AND WORD#16#FFEF;
       #H_HMI5ModeCmd := #H_HMI5ModeCmd AND WORD#16#FFEF;
   END_IF;
END_REGION

REGION Network 19: **** 1 - Inputs **** Set Auto select on HMI1 if plc go from STOP to RUN
   // Set Auto select on HMI1 if it´s not used
   IF "FirstScan" THEN #H_HMI1ModeCmd.%X0 := TRUE; END_IF;
END_REGION

REGION Network 20: **** 1 - Inputs **** Set Auto select on HMI2 if it´s not used or plc go from STOP to RUN
   // Set Auto select on HMI2 if it´s not used
   IF (#I_NumHMI < 2) OR "FirstScan" THEN #H_HMI2ModeCmd.%X0 := TRUE; END_IF;
END_REGION

REGION Network 21: **** 1 - Inputs **** Set Auto select on HMI3 if it´s not used or plc go from STOP to RUN
   // Set Auto select on HMI3 if it´s not used
   IF (#I_NumHMI < 3) OR "FirstScan" THEN #H_HMI3ModeCmd.%X0 := TRUE; END_IF;
END_REGION

REGION Network 22: **** 1 - Inputs **** Set Auto select on HMI4 if it´s not used or plc go from STOP to RUN
   // Set Auto select on HMI4 if it´s not used
   IF (#I_NumHMI < 4) OR "FirstScan" THEN #H_HMI4ModeCmd.%X0 := TRUE; END_IF;
END_REGION

REGION Network 23: **** 1 - Inputs **** Set Auto select on HMI5 if it´s not used or plc go from STOP to RUN
   // Set Auto select on HMI5 if it´s not used
   IF (#I_NumHMI < 5) OR "FirstScan" THEN #H_HMI5ModeCmd.%X0 := TRUE; END_IF;
END_REGION

REGION Network 24: **** 4.3 - Machine Status - Operator Sel **** Forced manual is selected on the active HMI
   // Forced manual is selected on the active HMI
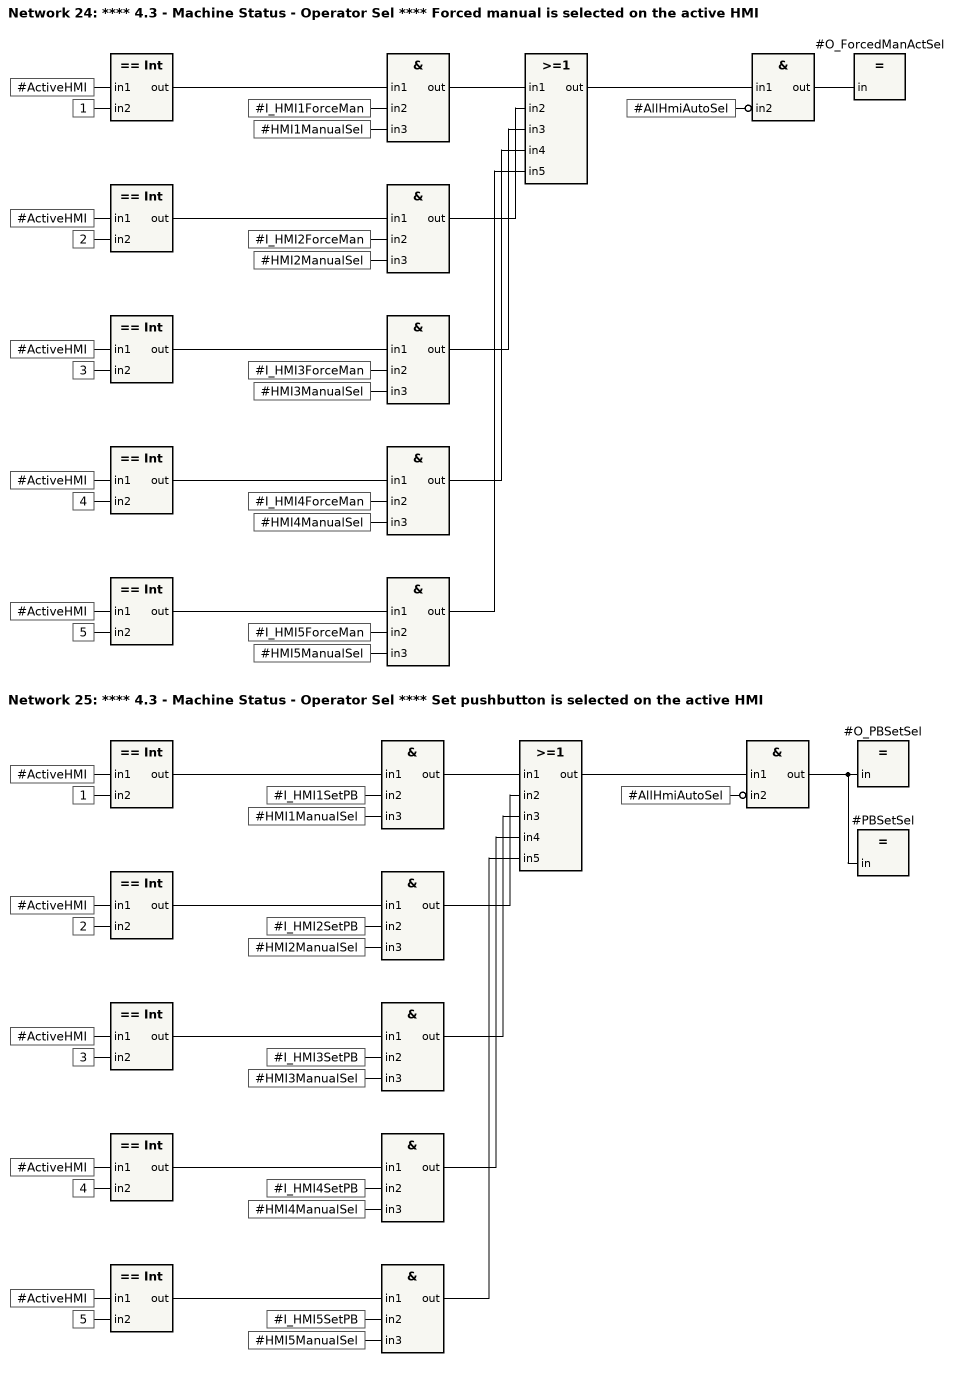
   #O_ForcedManActSel := (((#ActiveHMI = 1) AND #I_HMI1ForceMan AND #HMI1ManualSel) OR ((#ActiveHMI = 2) AND #I_HMI2ForceMan AND #HMI2ManualSel) OR ((#ActiveHMI = 3) AND #I_HMI3ForceMan AND #HMI3ManualSel) OR ((#ActiveHMI = 4) AND #I_HMI4ForceMan AND #HMI4ManualSel) OR ((#ActiveHMI = 5) AND #I_HMI5ForceMan AND #HMI5ManualSel)) AND NOT #AllHmiAutoSel;
END_REGION

REGION Network 25: **** 4.3 - Machine Status - Operator Sel **** Set pushbutton is selected on the active HMI
   // Set pushbutton is selected on the active HMI
   #O_PBSetSel := (((#ActiveHMI = 1) AND #I_HMI1SetPB AND #HMI1ManualSel) OR ((#ActiveHMI = 2) AND #I_HMI2SetPB AND #HMI2ManualSel) OR ((#ActiveHMI = 3) AND #I_HMI3SetPB AND #HMI3ManualSel) OR ((#ActiveHMI = 4) AND #I_HMI4SetPB AND #HMI4ManualSel) OR ((#ActiveHMI = 5) AND #I_HMI5SetPB AND #HMI5ManualSel)) AND NOT #AllHmiAutoSel;
   #PBSetSel := #O_PBSetSel;
END_REGION

REGION Network 26: **** 4.3 - Machine Status - Operator Sel **** Reset pushbutton is selected on the active HMI
   // Reset pushbutton is selected on the active HMI
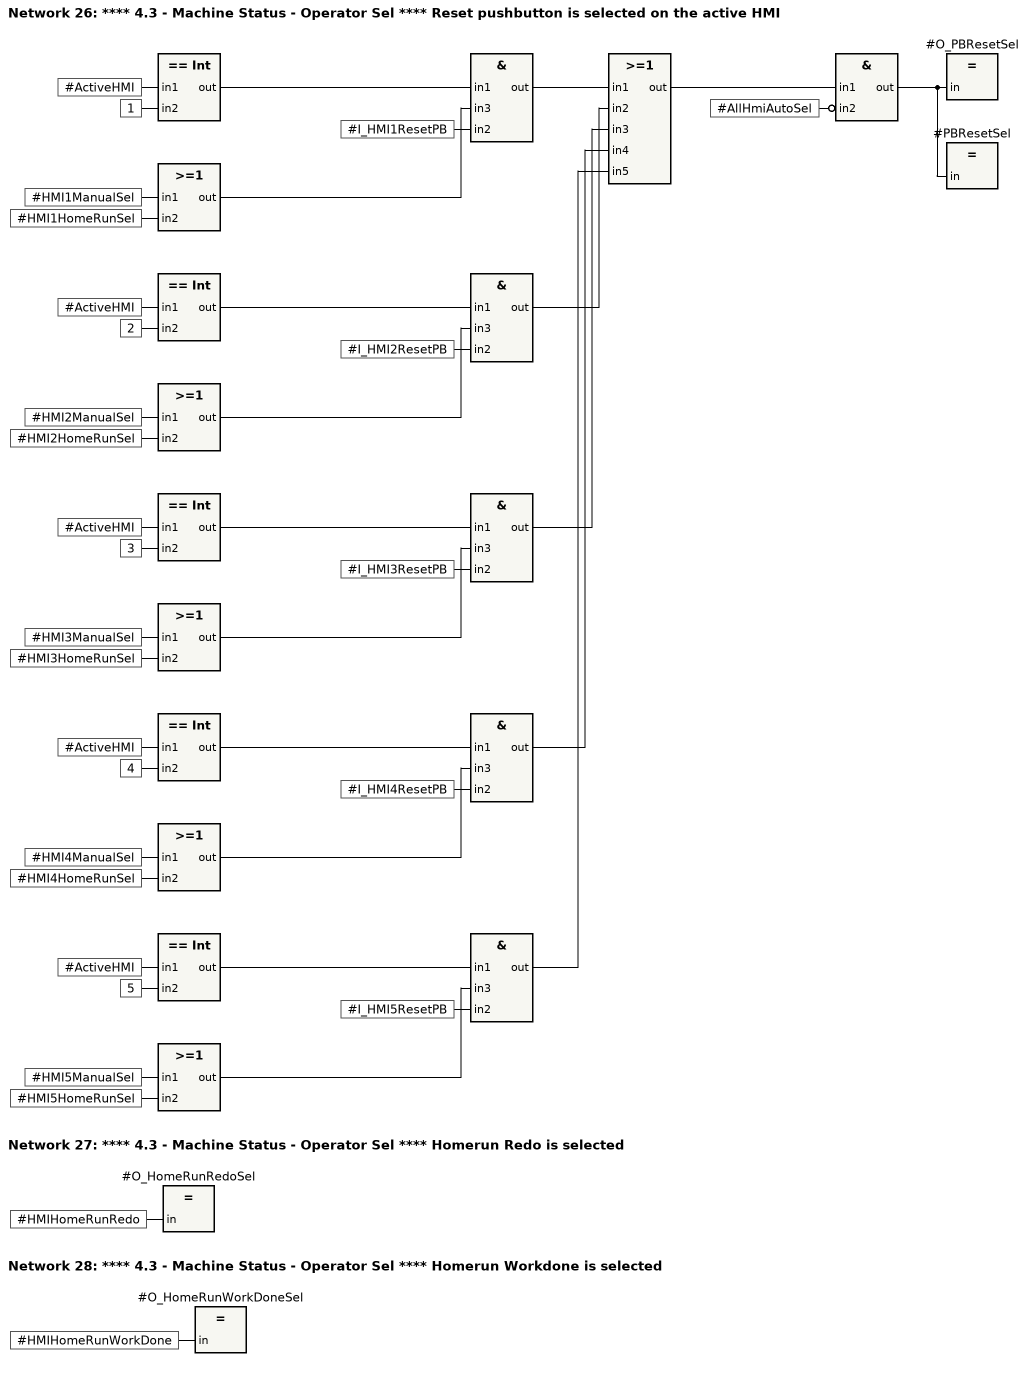
   #O_PBResetSel := (((#ActiveHMI = 1) AND (#HMI1ManualSel OR #HMI1HomeRunSel) AND #I_HMI1ResetPB) OR ((#ActiveHMI = 2) AND (#HMI2ManualSel OR #HMI2HomeRunSel) AND #I_HMI2ResetPB) OR ((#ActiveHMI = 3) AND (#HMI3ManualSel OR #HMI3HomeRunSel) AND #I_HMI3ResetPB) OR ((#ActiveHMI = 4) AND (#HMI4ManualSel OR #HMI4HomeRunSel) AND #I_HMI4ResetPB) OR ((#ActiveHMI = 5) AND (#HMI5ManualSel OR #HMI5HomeRunSel) AND #I_HMI5ResetPB)) AND NOT #AllHmiAutoSel;
   #PBResetSel := #O_PBResetSel;
END_REGION

REGION Network 27: **** 4.3 - Machine Status - Operator Sel **** Homerun Redo is selected
   // Homerun Redo is selected
   #O_HomeRunRedoSel := #HMIHomeRunRedo;
END_REGION

REGION Network 28: **** 4.3 - Machine Status - Operator Sel **** Homerun Workdone is selected
   // Homerun Workdone is selected
   #O_HomeRunWorkDoneSel := #HMIHomeRunWorkDone;
END_REGION

REGION Network 29: **** 4.4 - Machine Status - Calculated **** Lock manual button
   // Lock manual button
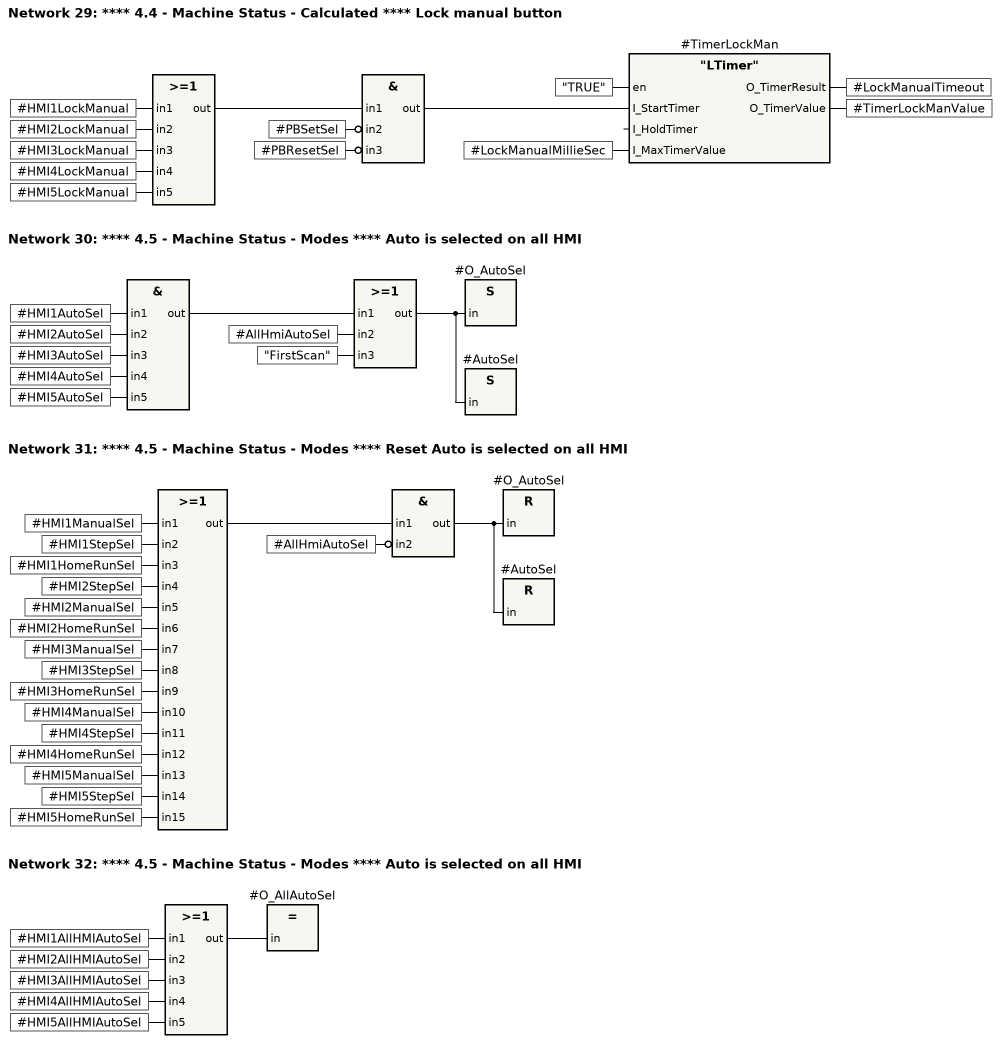
   IF "TRUE" THEN
       #TimerLockMan(I_StartTimer := (#HMI1LockManual OR #HMI2LockManual OR #HMI3LockManual OR #HMI4LockManual OR #HMI5LockManual) AND NOT #PBSetSel AND NOT #PBResetSel,   // "LTimer"
                     I_MaxTimerValue := #LockManualMillieSec,
                     O_TimerResult => #LockManualTimeout,
                     O_TimerValue => #TimerLockManValue);
   END_IF;
END_REGION

REGION Network 30: **** 4.5 - Machine Status - Modes **** Auto is selected on all HMI
   // Auto is selected on all HMI
   IF (#HMI1AutoSel AND #HMI2AutoSel AND #HMI3AutoSel AND #HMI4AutoSel AND #HMI5AutoSel) OR #AllHmiAutoSel OR "FirstScan" THEN
       #O_AutoSel := TRUE;
       #AutoSel := TRUE;
   END_IF;
END_REGION

REGION Network 31: **** 4.5 - Machine Status - Modes **** Reset Auto is selected on all HMI
   // Reset Auto is selected on all HMI
   IF (#HMI1ManualSel OR #HMI1StepSel OR #HMI1HomeRunSel OR #HMI2StepSel OR #HMI2ManualSel OR #HMI2HomeRunSel OR #HMI3ManualSel OR #HMI3StepSel OR #HMI3HomeRunSel OR #HMI4ManualSel OR #HMI4StepSel OR #HMI4HomeRunSel OR #HMI5ManualSel OR #HMI5StepSel OR #HMI5HomeRunSel) AND NOT #AllHmiAutoSel THEN
       #O_AutoSel := FALSE;
       #AutoSel := FALSE;
   END_IF;
END_REGION

REGION Network 32: **** 4.5 - Machine Status - Modes **** Auto is selected on all HMI
   // Auto is selected on all HMI
   #O_AllAutoSel := #HMI1AllHMIAutoSel OR #HMI2AllHMIAutoSel OR #HMI3AllHMIAutoSel OR #HMI4AllHMIAutoSel OR #HMI5AllHMIAutoSel;
END_REGION

REGION Network 33: **** 4.5 - Machine Status - Modes **** Step is selected on one HMI, the other HMI have auto selected
   // Step is selected on one HMI, the other HMI have auto selected
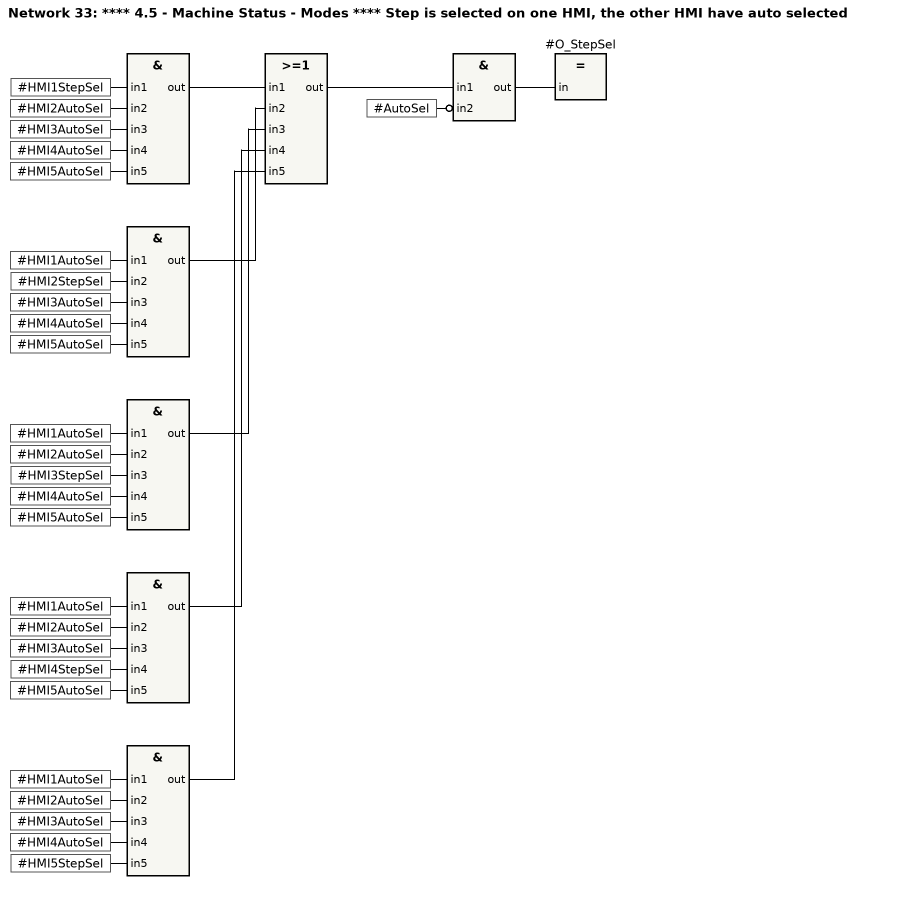
   #O_StepSel := ((#HMI1StepSel AND #HMI2AutoSel AND #HMI3AutoSel AND #HMI4AutoSel AND #HMI5AutoSel) OR (#HMI1AutoSel AND #HMI2StepSel AND #HMI3AutoSel AND #HMI4AutoSel AND #HMI5AutoSel) OR (#HMI1AutoSel AND #HMI2AutoSel AND #HMI3StepSel AND #HMI4AutoSel AND #HMI5AutoSel) OR (#HMI1AutoSel AND #HMI2AutoSel AND #HMI3AutoSel AND #HMI4StepSel AND #HMI5AutoSel) OR (#HMI1AutoSel AND #HMI2AutoSel AND #HMI3AutoSel AND #HMI4AutoSel AND #HMI5StepSel)) AND NOT #AutoSel;
END_REGION

REGION Network 34: **** 4.5 - Machine Status - Modes **** Homerun is selected on one HMI, the other HMI have auto selected
   // Homerun is selected on one HMI, the other HMI have auto selected
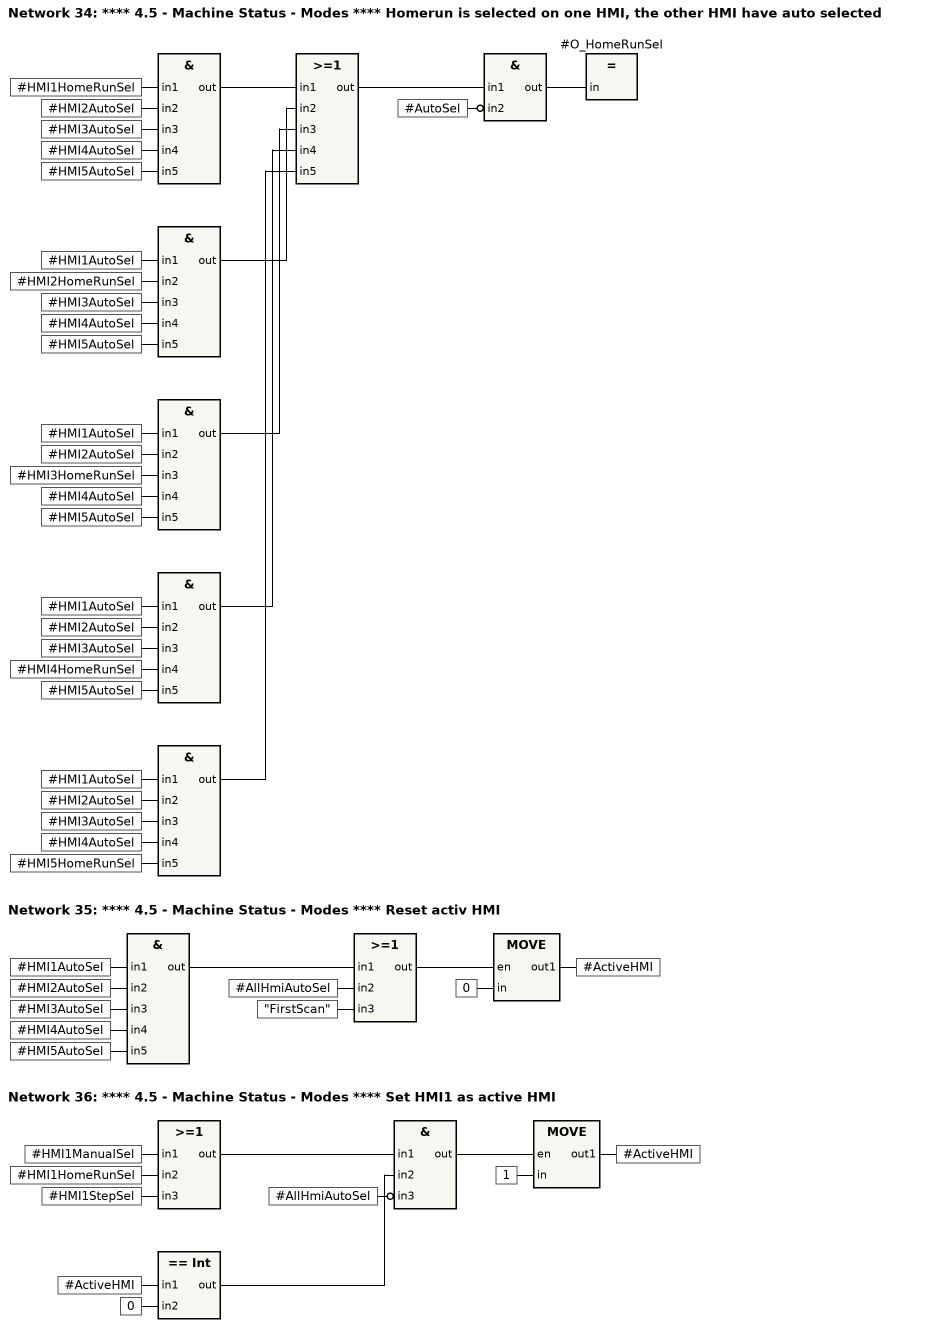
   #O_HomeRunSel := ((#HMI1HomeRunSel AND #HMI2AutoSel AND #HMI3AutoSel AND #HMI4AutoSel AND #HMI5AutoSel) OR (#HMI1AutoSel AND #HMI2HomeRunSel AND #HMI3AutoSel AND #HMI4AutoSel AND #HMI5AutoSel) OR (#HMI1AutoSel AND #HMI2AutoSel AND #HMI3HomeRunSel AND #HMI4AutoSel AND #HMI5AutoSel) OR (#HMI1AutoSel AND #HMI2AutoSel AND #HMI3AutoSel AND #HMI4HomeRunSel AND #HMI5AutoSel) OR (#HMI1AutoSel AND #HMI2AutoSel AND #HMI3AutoSel AND #HMI4AutoSel AND #HMI5HomeRunSel)) AND NOT #AutoSel;
END_REGION

REGION Network 35: **** 4.5 - Machine Status - Modes **** Reset activ HMI
   // Reset activ HMI
   IF (#HMI1AutoSel AND #HMI2AutoSel AND #HMI3AutoSel AND #HMI4AutoSel AND #HMI5AutoSel) OR #AllHmiAutoSel OR "FirstScan" THEN
       #ActiveHMI := 0;
   END_IF;
END_REGION

REGION Network 36: **** 4.5 - Machine Status - Modes **** Set HMI1 as active HMI
   // Set HMI1 as active HMI
   IF (#HMI1ManualSel OR #HMI1HomeRunSel OR #HMI1StepSel) AND (#ActiveHMI = 0) AND NOT #AllHmiAutoSel THEN
       #ActiveHMI := 1;
   END_IF;
END_REGION

REGION Network 37: **** 4.5 - Machine Status - Modes **** Set HMI2 as active HMI
   // Set HMI2 as active HMI
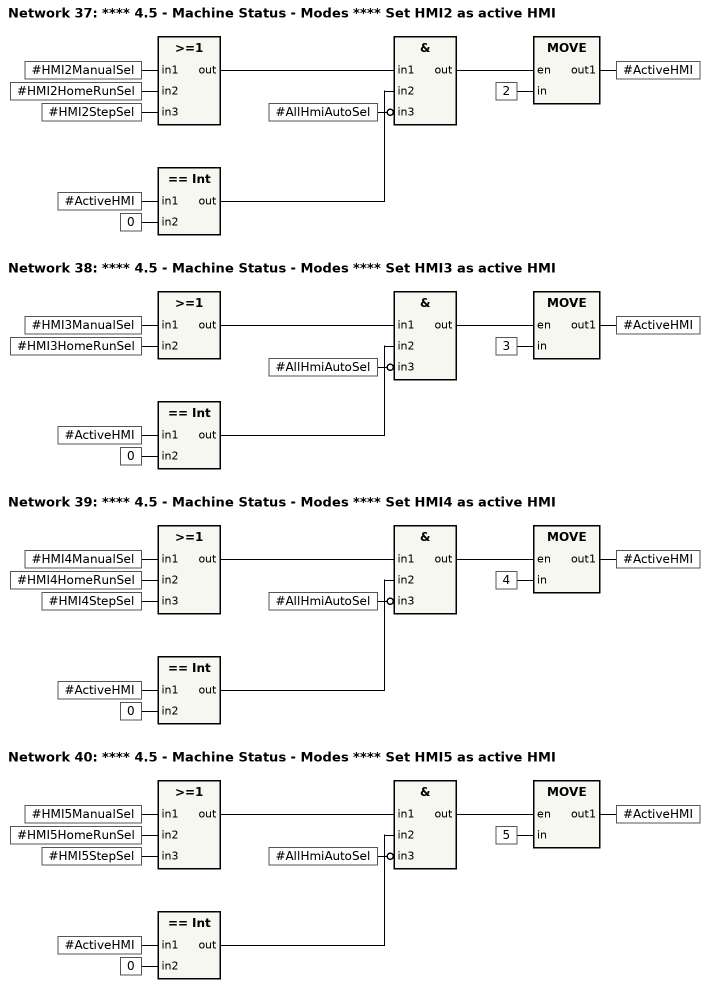
   IF (#HMI2ManualSel OR #HMI2HomeRunSel OR #HMI2StepSel) AND (#ActiveHMI = 0) AND NOT #AllHmiAutoSel THEN
       #ActiveHMI := 2;
   END_IF;
END_REGION

REGION Network 38: **** 4.5 - Machine Status - Modes **** Set HMI3 as active HMI
   // Set HMI3 as active HMI
   IF (#HMI3ManualSel OR #HMI3HomeRunSel) AND (#ActiveHMI = 0) AND NOT #AllHmiAutoSel THEN
       #ActiveHMI := 3;
   END_IF;
END_REGION

REGION Network 39: **** 4.5 - Machine Status - Modes **** Set HMI4 as active HMI
   // Set HMI4 as active HMI
   IF (#HMI4ManualSel OR #HMI4HomeRunSel OR #HMI4StepSel) AND (#ActiveHMI = 0) AND NOT #AllHmiAutoSel THEN
       #ActiveHMI := 4;
   END_IF;
END_REGION

REGION Network 40: **** 4.5 - Machine Status - Modes **** Set HMI5 as active HMI
   // Set HMI5 as active HMI
   IF (#HMI5ManualSel OR #HMI5HomeRunSel OR #HMI5StepSel) AND (#ActiveHMI = 0) AND NOT #AllHmiAutoSel THEN
       #ActiveHMI := 5;
   END_IF;
END_REGION

REGION Network 41: **** 4.5 - Machine Status - Modes **** Set Manual selected if one of the HMI is active
   // Set Manual selected if one of the HMI is active
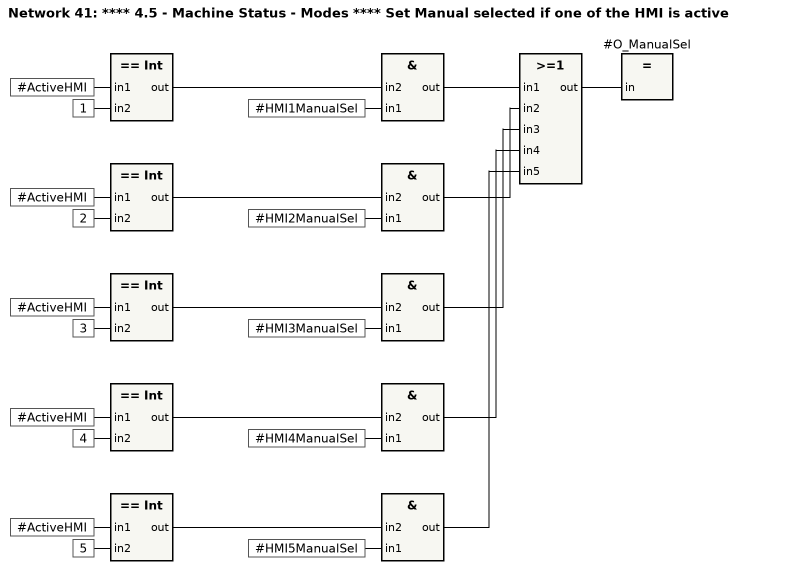
   #O_ManualSel := ((#ActiveHMI = 1) AND #HMI1ManualSel) OR ((#ActiveHMI = 2) AND #HMI2ManualSel) OR ((#ActiveHMI = 3) AND #HMI3ManualSel) OR ((#ActiveHMI = 4) AND #HMI4ManualSel) OR ((#ActiveHMI = 5) AND #HMI5ManualSel);
END_REGION

REGION Network 42: **** 4.6 - Machine Status - Indications **** Animation
   // Animation
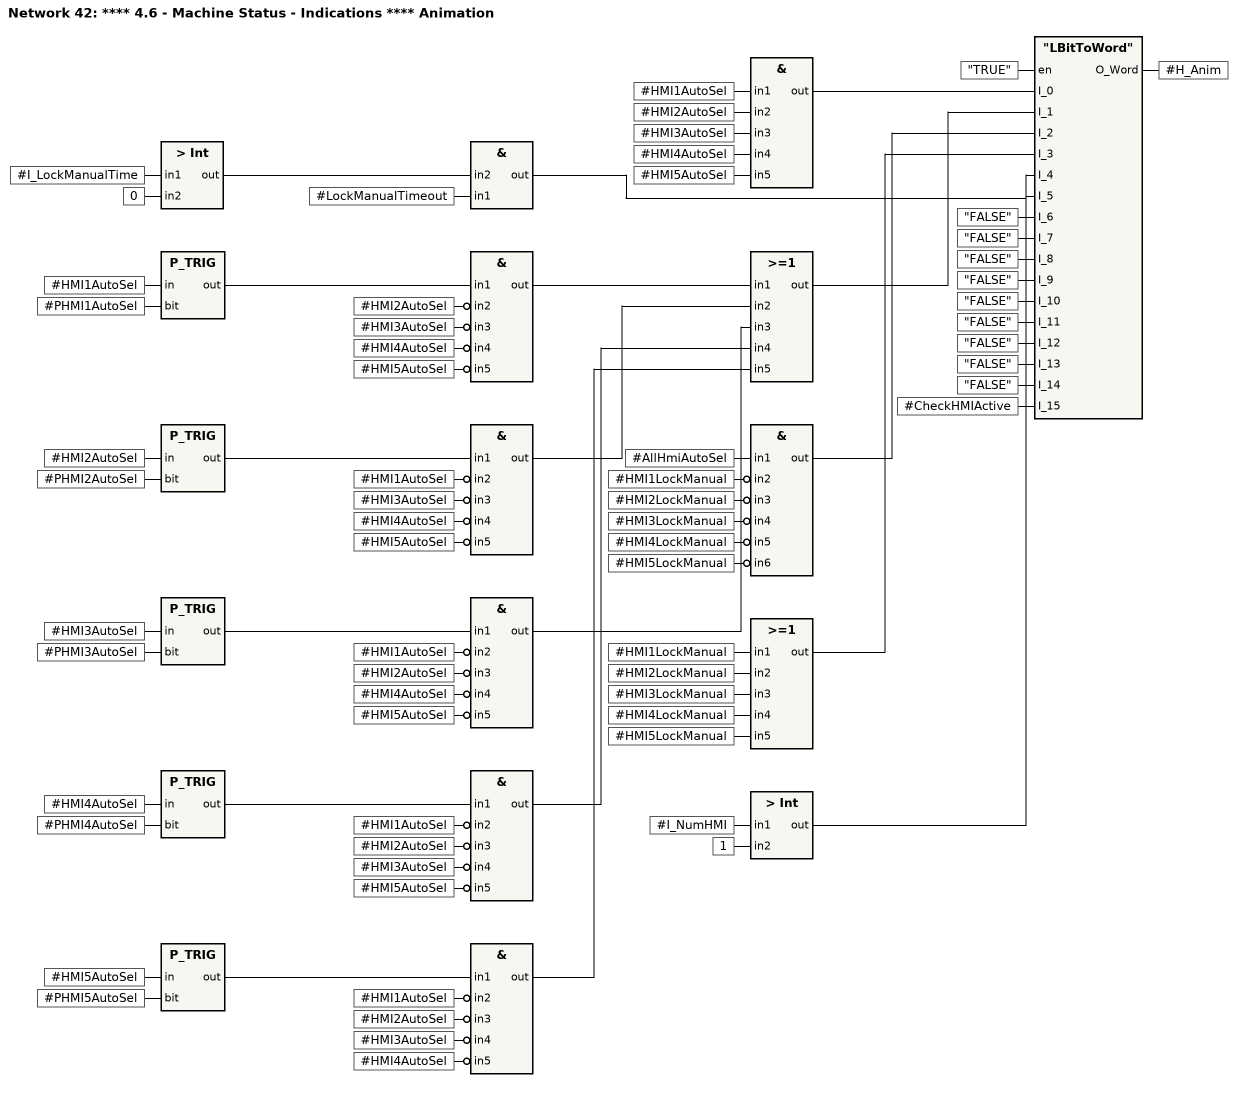
   #_w1 := #HMI1AutoSel AND NOT #PHMI1AutoSel;   // rising edge
   #PHMI1AutoSel := #HMI1AutoSel;
   #_w2 := #HMI2AutoSel AND NOT #PHMI2AutoSel;   // rising edge
   #PHMI2AutoSel := #HMI2AutoSel;
   #_w3 := #HMI3AutoSel AND NOT #PHMI3AutoSel;   // rising edge
   #PHMI3AutoSel := #HMI3AutoSel;
   #_w4 := #HMI4AutoSel AND NOT #PHMI4AutoSel;   // rising edge
   #PHMI4AutoSel := #HMI4AutoSel;
   #_w5 := #HMI5AutoSel AND NOT #PHMI5AutoSel;   // rising edge
   #PHMI5AutoSel := #HMI5AutoSel;
   IF "TRUE" THEN
       "LBitToWord"(I_0 := #HMI1AutoSel AND #HMI2AutoSel AND #HMI3AutoSel AND #HMI4AutoSel AND #HMI5AutoSel,
                    I_1 := (#_w1 AND NOT #HMI2AutoSel AND NOT #HMI3AutoSel AND NOT #HMI4AutoSel AND NOT #HMI5AutoSel) OR (#_w2 AND NOT #HMI1AutoSel AND NOT #HMI3AutoSel AND NOT #HMI4AutoSel AND NOT #HMI5AutoSel) OR (#_w3 AND NOT #HMI1AutoSel AND NOT #HMI2AutoSel AND NOT #HMI4AutoSel AND NOT #HMI5AutoSel) OR (#_w4 AND NOT #HMI1AutoSel AND NOT #HMI2AutoSel AND NOT #HMI3AutoSel AND NOT #HMI5AutoSel) OR (#_w5 AND NOT #HMI1AutoSel AND NOT #HMI2AutoSel AND NOT #HMI3AutoSel AND NOT #HMI4AutoSel),
                    I_2 := #AllHmiAutoSel AND NOT #HMI1LockManual AND NOT #HMI2LockManual AND NOT #HMI3LockManual AND NOT #HMI4LockManual AND NOT #HMI5LockManual,
                    I_3 := #HMI1LockManual OR #HMI2LockManual OR #HMI3LockManual OR #HMI4LockManual OR #HMI5LockManual,
                    I_4 := (#I_LockManualTime > 0) AND #LockManualTimeout,
                    I_5 := #I_NumHMI > 1,
                    I_6 := "FALSE",
                    I_7 := "FALSE",
                    I_8 := "FALSE",
                    I_9 := "FALSE",
                    I_10 := "FALSE",
                    I_11 := "FALSE",
                    I_12 := "FALSE",
                    I_13 := "FALSE",
                    I_14 := "FALSE",
                    I_15 := #CheckHMIActive,
                    O_Word => #H_Anim);
   END_IF;
END_REGION

REGION Network 43: **** 5.2 - Equations - Flow **** Reset transport memory on active HMI
   // Reset transport memory on active HMI
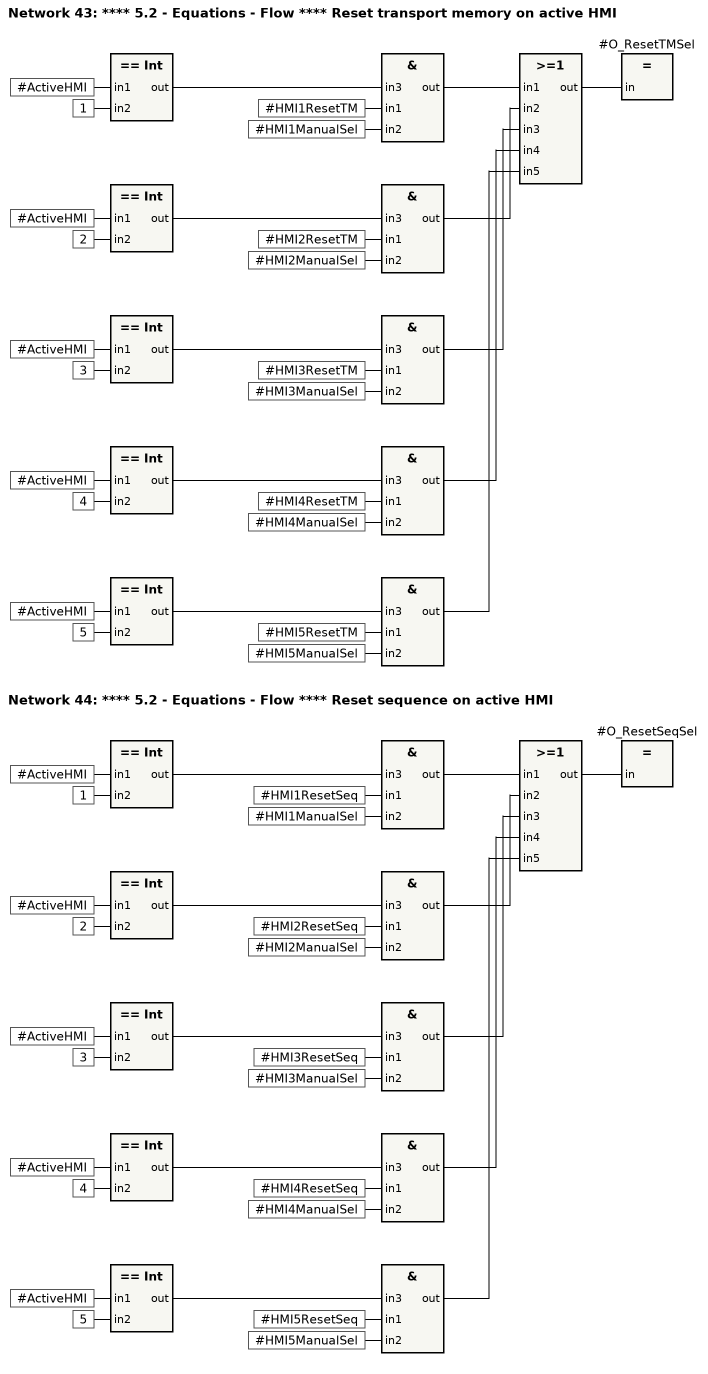
   #O_ResetTMSel := ((#ActiveHMI = 1) AND #HMI1ResetTM AND #HMI1ManualSel) OR ((#ActiveHMI = 2) AND #HMI2ResetTM AND #HMI2ManualSel) OR ((#ActiveHMI = 3) AND #HMI3ResetTM AND #HMI3ManualSel) OR ((#ActiveHMI = 4) AND #HMI4ResetTM AND #HMI4ManualSel) OR ((#ActiveHMI = 5) AND #HMI5ResetTM AND #HMI5ManualSel);
END_REGION

REGION Network 44: **** 5.2 - Equations - Flow **** Reset sequence on active HMI
   // Reset sequence on active HMI
   #O_ResetSeqSel := ((#ActiveHMI = 1) AND #HMI1ResetSeq AND #HMI1ManualSel) OR ((#ActiveHMI = 2) AND #HMI2ResetSeq AND #HMI2ManualSel) OR ((#ActiveHMI = 3) AND #HMI3ResetSeq AND #HMI3ManualSel) OR ((#ActiveHMI = 4) AND #HMI4ResetSeq AND #HMI4ManualSel) OR ((#ActiveHMI = 5) AND #HMI5ResetSeq AND #HMI5ManualSel);
END_REGION

REGION Network 45: **** 5.2 - Equations - Flow **** Reset Failsafe reset register
   // Reset Failsafe reset register
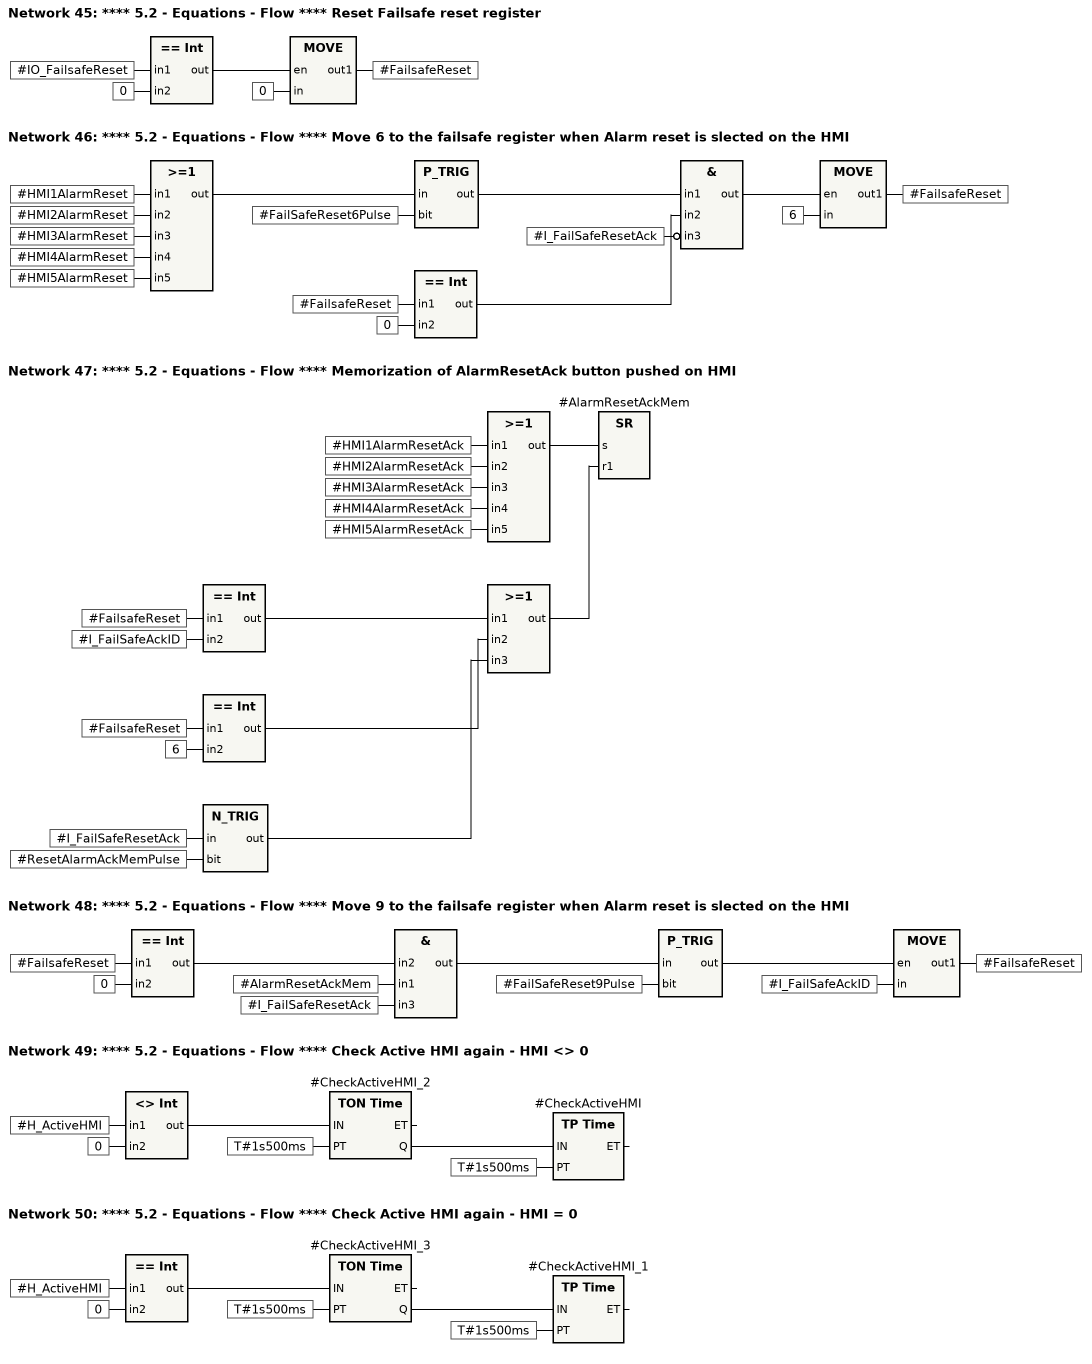
   IF #IO_FailsafeReset = 0 THEN #FailsafeReset := 0; END_IF;
END_REGION

REGION Network 46: **** 5.2 - Equations - Flow **** Move 6 to the failsafe register when Alarm reset is slected on the HMI
   // Move 6 to the failsafe register when Alarm reset is slected on the HMI
   #_w1 := #HMI1AlarmReset OR #HMI2AlarmReset OR #HMI3AlarmReset OR #HMI4AlarmReset OR #HMI5AlarmReset;
   #_w2 := #_w1 AND NOT #FailSafeReset6Pulse;   // rising edge
   #FailSafeReset6Pulse := #_w1;
   IF #_w2 AND (#FailsafeReset = 0) AND NOT #I_FailSafeResetAck THEN #FailsafeReset := 6; END_IF;
END_REGION

REGION Network 47: **** 5.2 - Equations - Flow **** Memorization of AlarmResetAck button pushed on HMI
   // Memorization of AlarmResetAck button pushed on HMI
   #_w1 := NOT #I_FailSafeResetAck AND #ResetAlarmAckMemPulse;   // falling edge
   #ResetAlarmAckMemPulse := #I_FailSafeResetAck;
   IF #HMI1AlarmResetAck OR #HMI2AlarmResetAck OR #HMI3AlarmResetAck OR #HMI4AlarmResetAck OR #HMI5AlarmResetAck THEN
       #AlarmResetAckMem := TRUE;   // SR flip-flop
   END_IF;
   IF (#FailsafeReset = #I_FailSafeAckID) OR (#FailsafeReset = 6) OR #_w1 THEN
       #AlarmResetAckMem := FALSE;
   END_IF;
END_REGION

REGION Network 48: **** 5.2 - Equations - Flow **** Move 9 to the failsafe register when Alarm reset is slected on the HMI
   // Move 9 to the failsafe register when Alarm reset is slected on the HMI
   #_w1 := (#FailsafeReset = 0) AND #AlarmResetAckMem AND #I_FailSafeResetAck;
   #_w2 := #_w1 AND NOT #FailSafeReset9Pulse;   // rising edge
   #FailSafeReset9Pulse := #_w1;
   IF #_w2 THEN #FailsafeReset := #I_FailSafeAckID; END_IF;
END_REGION

REGION Network 49: **** 5.2 - Equations - Flow **** Check Active HMI again - HMI <> 0
   // Check Active HMI again
   #CheckActiveHMI_2(IN := #H_ActiveHMI <> 0, PT := T#1s500ms);   // TON
   #CheckActiveHMI(IN := #CheckActiveHMI_2.Q, PT := T#1s500ms);   // TP
END_REGION

REGION Network 50: **** 5.2 - Equations - Flow **** Check Active HMI again - HMI = 0
   // Check Active HMI again
   #CheckActiveHMI_3(IN := #H_ActiveHMI = 0, PT := T#1s500ms);   // TON
   #CheckActiveHMI_1(IN := #CheckActiveHMI_3.Q, PT := T#1s500ms);   // TP
END_REGION

REGION Network 51: **** 5.2 - Equations - Flow **** Check Active HMI
   // Check Active HMI
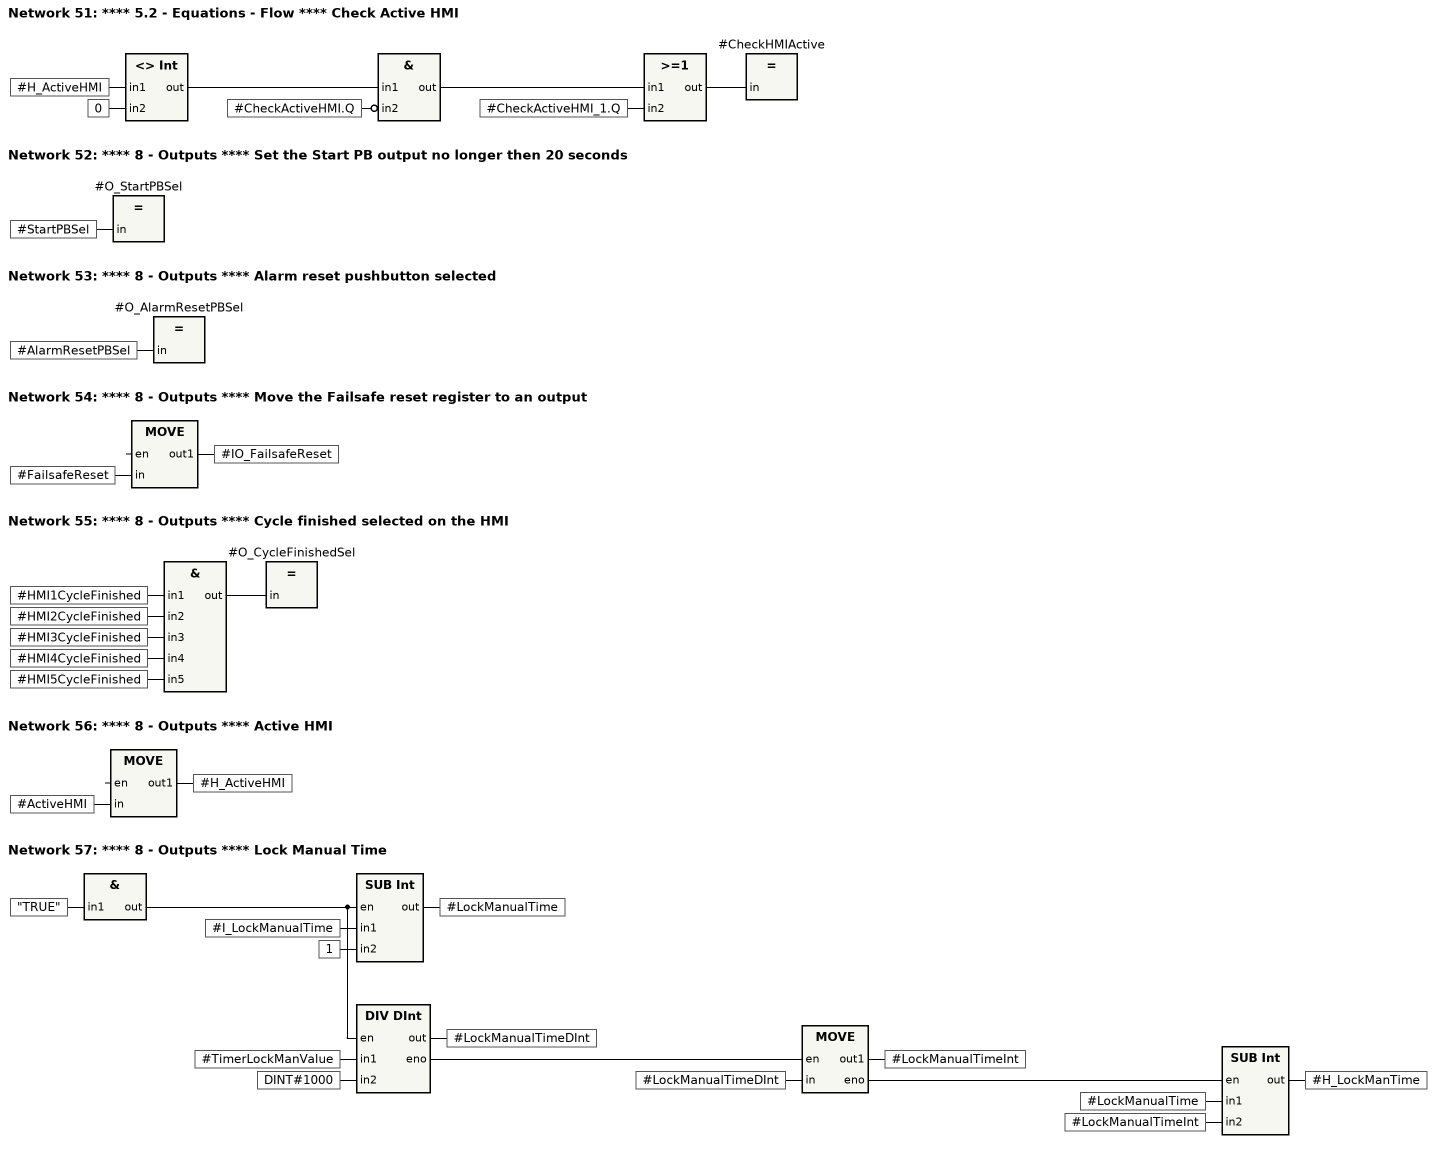
   #CheckHMIActive := ((#H_ActiveHMI <> 0) AND NOT #CheckActiveHMI.Q) OR #CheckActiveHMI_1.Q;
END_REGION

REGION Network 52: **** 8 - Outputs **** Set the Start PB output no longer then 20 seconds
   // Set the Start PB output no longer then 20 seconds
   #O_StartPBSel := #StartPBSel;
END_REGION

REGION Network 53: **** 8 - Outputs **** Alarm reset pushbutton selected
   // Alarm reset pushbutton selected
   #O_AlarmResetPBSel := #AlarmResetPBSel;
END_REGION

REGION Network 54: **** 8 - Outputs **** Move the Failsafe reset register to an output
   // Move the Failsafe reset register to an output
   #IO_FailsafeReset := #FailsafeReset;
END_REGION

REGION Network 55: **** 8 - Outputs **** Cycle finished selected on the HMI
   // Cycle finished selected on the HMI
   #O_CycleFinishedSel := #HMI1CycleFinished AND #HMI2CycleFinished AND #HMI3CycleFinished AND #HMI4CycleFinished AND #HMI5CycleFinished;
END_REGION

REGION Network 56: **** 8 - Outputs **** Active HMI
   // Active HMI
   #H_ActiveHMI := #ActiveHMI;
END_REGION

REGION Network 57: **** 8 - Outputs **** Lock Manual Time
   // Lock Manual Time
   // ENO of a box is taken as its EN; it also drops when the box reports an error
   IF "TRUE" THEN
       #LockManualTime := #I_LockManualTime - 1;
       #LockManualTimeDInt := #TimerLockManValue / DINT#1000;
       #LockManualTimeInt := #LockManualTimeDInt;
       #H_LockManTime := #LockManualTime - #LockManualTimeInt;
   END_IF;
END_REGION
END_FUNCTION_BLOCK
